	(* conversion string to value *)
		i:=1;
		(* read string line-->Group or NodeId *)
		sTmp:=T_Axis.T_FileObj.sData[i];
		iPosCarStart:=FIND(sTmp,':=')+2;
		iPosCarStop:=FIND(sTmp,';');
		IF ((iPosCarStart - 2) = 0) OR (iPosCarStop = 0) OR (iPosCarStart >= iPosCarStop) THEN xBusy:=FALSE;	xDone:=FALSE; xError:=TRUE; diErrorNr:=16#F100;	(* Wrong Syntax from Axis File *) RETURN; END_IF;
		T_Axis.T_Config_Gen.udiNC_TaskIdxGrp:=0;
		T_Axis.T_Config_Gen.udiNodeId:=STRING_TO_UDINT(MID(sTmp,iPosCarStop-iPosCarStart,iPosCarStart));
		i:=i+1;
		(* read string line-->ADS NetID *)
		sTmp:=T_Axis.T_FileObj.sData[i];
		iPosCarStart:=FIND(sTmp,':=')+2;
		iPosCarStop:=FIND(sTmp,';');
		IF ((iPosCarStart - 2) = 0) OR (iPosCarStop = 0) OR (iPosCarStart >= iPosCarStop) THEN xBusy:=FALSE;	xDone:=FALSE; xError:=TRUE; diErrorNr:=16#F100;	(* Wrong Syntax from Axis File *) RETURN; END_IF;
		T_Axis.T_Config_Gen.sServoNetId:='';
		T_Axis.T_Config_Gen.sAmsNetId:=MID(sTmp,iPosCarStop-iPosCarStart,iPosCarStart);
		i:=i+1;
		(* read string line-->DeviceName *)
		sTmp:=T_Axis.T_FileObj.sData[i];
		iPosCarStart:=FIND(sTmp,':=')+2;
   		iPosCarStop:=FIND(sTmp,';');
		IF ((iPosCarStart - 2) = 0) OR (iPosCarStop = 0) OR (iPosCarStart >= iPosCarStop) THEN xBusy:=FALSE;	xDone:=FALSE; xError:=TRUE; diErrorNr:=16#F100;	(* Wrong Syntax from Axis File *) RETURN; END_IF;
		T_Axis.T_Config_Gen.sFileNamePDOMapping:=MID(sTmp,iPosCarStop-iPosCarStart,iPosCarStart);
		i:=i+1;
		jj:=1;
		(* read string lines *)
		WHILE T_Axis.T_FileObj.sData[i] <> '' DO
			sTmp:=T_Axis.T_FileObj.sData[i];
			(* index group *)
			iPosCarStart:=FIND(sTmp,':=')+2;
			iPosCarStop:=FIND(sTmp,';');
			IF ((iPosCarStart - 2) = 0) OR (iPosCarStop = 0) OR (iPosCarStart >= iPosCarStop) THEN xBusy:=FALSE;	xDone:=FALSE; xError:=TRUE; diErrorNr:=16#F100;	(* Wrong Syntax from Axis File *) RETURN; END_IF;
			T_Axis.T_ParamFileObj[jj].udiIdxGroup:=	STRING_TO_UDINT(MID(sTmp,iPosCarStop-iPosCarStart,iPosCarStart))
											+ T_Axis.T_Config_Gen.udiNC_TaskIdxGrp;
			sTmp:=MID(sTmp,LEN(sTmp)-iPosCarStop, iPosCarStop+1);
			(* index offset *)
			iPosCarStart:=FIND(sTmp,':=')+2;
			iPosCarStop:=FIND(sTmp,';');
			IF ((iPosCarStart - 2) = 0) OR (iPosCarStop = 0) OR (iPosCarStart >= iPosCarStop) THEN xBusy:=FALSE;	xDone:=FALSE; xError:=TRUE; diErrorNr:=16#F100;	(* Wrong Syntax from Axis File *) RETURN; END_IF;
			T_Axis.T_ParamFileObj[jj].udiIndexOffset:=STRING_TO_UDINT(MID(sTmp,iPosCarStop-iPosCarStart,iPosCarStart));
			sTmp:=MID(sTmp,LEN(sTmp)-iPosCarStop, iPosCarStop+1);
			(* length value *)
			iPosCarStart:=FIND(sTmp,':=')+2;
			iPosCarStop:=FIND(sTmp,';');
			IF ((iPosCarStart - 2) = 0) OR (iPosCarStop = 0) OR (iPosCarStart >= iPosCarStop) THEN xBusy:=FALSE;	xDone:=FALSE; xError:=TRUE; diErrorNr:=16#F100;	(* Wrong Syntax from Axis File *) RETURN; END_IF;
			T_Axis.T_ParamFileObj[jj].udiLength:=STRING_TO_UDINT(MID(sTmp,iPosCarStop-iPosCarStart,iPosCarStart));
			sTmp:=MID(sTmp,LEN(sTmp)-iPosCarStop, iPosCarStop+1);
			(* value*)
			iPosCarStart:=FIND(sTmp,':=')+2;
			iPosCarStop:=FIND(sTmp,';');
			IF ((iPosCarStart - 2) = 0) OR (iPosCarStop = 0) OR (iPosCarStart >= iPosCarStop) THEN xBusy:=FALSE;	xDone:=FALSE; xError:=TRUE; diErrorNr:=16#F100;	(* Wrong Syntax from Axis File *) RETURN; END_IF;
			T_Axis.T_ParamFileObj[jj].lrReal:=UDINT_TO_REAL(STRING_TO_UDINT(MID(sTmp,iPosCarStop-iPosCarStart,iPosCarStart)));
			(* init existing line, erase text *)
			iPosCarStop:=FIND(T_Axis.T_FileObj.sData[i],'(');
			T_Axis.T_FileObj.sData[i]:=MID(T_Axis.T_FileObj.sData[i],iPosCarStop-1,1);
			(* next line *)
			i:=i+1;
			jj:=jj+1;
		END_WHILE
		(* init. next *)
		T_Axis.T_ParamFileObj[jj].udiIdxGroup:=0;
		T_Axis.T_ParamFileObj[jj].udiIndexOffset:=0;
		T_Axis.T_ParamFileObj[jj].udiLength:=0;
		T_Axis.T_ParamFileObj[jj].lrReal:=0;

		(* set flag done *)
		xBusy:=FALSE;
		xDone:=TRUE;
END_FUNCTION_BLOCK

(* POU FB_HARDWARE/FB_CONVERT_AXISPARAMETER, ST *)
FUNCTION_BLOCK FB_CONVERT_AXISPARAMETER
VAR_INPUT
	xStart:BOOL;
END_VAR
VAR_IN_OUT
	T_Axis:ST_AXIS;
END_VAR
VAR_OUTPUT
	xDone:BOOL;
	xBusy:BOOL;
	xError:BOOL;
	diErrorNr:DINT;
END_VAR
VAR
(* trigger *)
	RisingEdgeStart:R_TRIG;
(* variable *)
	i: INT;
	iPosCarStart,iPosCarStop:INT;
	iStepConvertValueString:INT;
(* tmp variable *)
	sTmp:STRING(255);
	jj: INT;
END_VAR
(****************************************************************************************************************************************************)
(***********                                    This Functionblock convert the axis parameter for the EcoStep drive                                       ************)
(****************************************************************************************************************************************************)
(* wait start *)
	RisingEdgeStart(CLK:=xStart);
	IF RisingEdgeStart.Q THEN
	(* init. varaible *)
		iStepConvertValueString:=1;
		xDone:=FALSE;
	(*activ busy flag*)
		xBusy:=TRUE;
		xError:=FALSE;
		diErrorNr:=0;
	END_IF

(* test if activ *)
	IF NOT(xBusy) THEN
	(* exit FB *)
		RETURN;
	END_IF

	(* conversion string to value *)
		i:=1;
		(* read string line-->Group or NodeId *)
		sTmp:=T_Axis.T_FileObj.sData[i];
		iPosCarStart:=FIND(sTmp,':=')+2;
		iPosCarStop:=FIND(sTmp,';');
		IF ((iPosCarStart - 2) = 0) OR (iPosCarStop = 0) OR (iPosCarStart >= iPosCarStop) THEN xBusy:=FALSE;	xDone:=FALSE; xError:=TRUE; diErrorNr:=16#F100;	(* Wrong Syntax from Axis File *) RETURN; END_IF;
		T_Axis.T_Config_Gen.udiNC_TaskIdxGrp:=0;
		T_Axis.T_Config_Gen.udiNodeId:=STRING_TO_UDINT(MID(sTmp,iPosCarStop-iPosCarStart,iPosCarStart));
		i:=i+1;
		(* read string line-->ADS NetID *)
		sTmp:=T_Axis.T_FileObj.sData[i];
		iPosCarStart:=FIND(sTmp,':=')+2;
		iPosCarStop:=FIND(sTmp,';');
		IF ((iPosCarStart - 2) = 0) OR (iPosCarStop = 0) OR (iPosCarStart >= iPosCarStop) THEN xBusy:=FALSE;	xDone:=FALSE; xError:=TRUE; diErrorNr:=16#F100;	(* Wrong Syntax from Axis File *) RETURN; END_IF;
		T_Axis.T_Config_Gen.sServoNetId:='';
		T_Axis.T_Config_Gen.sAmsNetId:=MID(sTmp,iPosCarStop-iPosCarStart,iPosCarStart);
		i:=i+1;
		(* read string line-->DeviceName *)
		sTmp:=T_Axis.T_FileObj.sData[i];
		iPosCarStart:=FIND(sTmp,':=')+2;
   		iPosCarStop:=FIND(sTmp,';');
		IF ((iPosCarStart - 2) = 0) OR (iPosCarStop = 0) OR (iPosCarStart >= iPosCarStop) THEN xBusy:=FALSE;	xDone:=FALSE; xError:=TRUE; diErrorNr:=16#F100;	(* Wrong Syntax from Axis File *) RETURN; END_IF;
		T_Axis.T_Config_Gen.sDeviceFileName:=MID(sTmp,iPosCarStop-iPosCarStart,iPosCarStart);
		i:=i+1;
		(* read string line-->Scalefactor *)
		sTmp:=T_Axis.T_FileObj.sData[i];
		iPosCarStart:=FIND(sTmp,':=')+2;
   		iPosCarStop:=FIND(sTmp,';');
		IF ((iPosCarStart - 2) = 0) OR (iPosCarStop = 0) OR (iPosCarStart >= iPosCarStop) THEN xBusy:=FALSE;	xDone:=FALSE; xError:=TRUE; diErrorNr:=16#F100;	(* Wrong Syntax from Axis File *) RETURN; END_IF;
		T_Axis.T_CtrleSingle.lrScaleFactor:=STRING_TO_LREAL(MID(sTmp,iPosCarStop-iPosCarStart,iPosCarStart));
		i:=i+1;
		(* read string line-->GearRatioFactor  *)
		sTmp:=T_Axis.T_FileObj.sData[i];
		iPosCarStart:=FIND(sTmp,':=')+2;
   		iPosCarStop:=FIND(sTmp,';');
		IF ((iPosCarStart - 2) = 0) OR (iPosCarStop = 0) OR (iPosCarStart >= iPosCarStop) THEN xBusy:=FALSE;	xDone:=FALSE; xError:=TRUE; diErrorNr:=16#F100;	(* Wrong Syntax from Axis File *) RETURN; END_IF;
		T_Axis.T_CtrleSingle.lrGearRatioFactor:=STRING_TO_LREAL(MID(sTmp,iPosCarStop-iPosCarStart,iPosCarStart));
		i:=i+1;
		(* read string line-->GearRatioDivider *)
		sTmp:=T_Axis.T_FileObj.sData[i];
		iPosCarStart:=FIND(sTmp,':=')+2;
   		iPosCarStop:=FIND(sTmp,';');
		IF ((iPosCarStart - 2) = 0) OR (iPosCarStop = 0) OR (iPosCarStart >= iPosCarStop) THEN xBusy:=FALSE;	xDone:=FALSE; xError:=TRUE; diErrorNr:=16#F100;	(* Wrong Syntax from Axis File *) RETURN; END_IF;
		T_Axis.T_CtrleSingle.lrGearRatioDivider:=STRING_TO_LREAL(MID(sTmp,iPosCarStop-iPosCarStart,iPosCarStart));
		IF (T_Axis.T_CtrleSingle.lrGearRatioFactor <> 0) AND (T_Axis.T_CtrleSingle.lrGearRatioDivider <> 0) THEN
			T_Axis.T_CtrleSingle.lrGearRatio:=T_Axis.T_CtrleSingle.lrGearRatioFactor/T_Axis.T_CtrleSingle.lrGearRatioDivider;
		ELSE
			T_Axis.T_CtrleSingle.lrGearRatio:=1;
		END_IF;
		i:=i+1;
		jj:=1;
		(* read string lines *)
		WHILE T_Axis.T_FileObj.sData[i] <> '' DO
			sTmp:=T_Axis.T_FileObj.sData[i];
			(* index group *)
			iPosCarStart:=FIND(sTmp,':=')+2;
			iPosCarStop:=FIND(sTmp,';');
			IF ((iPosCarStart - 2) = 0) OR (iPosCarStop = 0) OR (iPosCarStart >= iPosCarStop) THEN xBusy:=FALSE;	xDone:=FALSE; xError:=TRUE; diErrorNr:=16#F100;	(* Wrong Syntax from Axis File *) RETURN; END_IF;
			T_Axis.T_ParamFileObj[jj].udiIdxGroup:=	STRING_TO_UDINT(MID(sTmp,iPosCarStop-iPosCarStart,iPosCarStart))
											+ T_Axis.T_Config_Gen.udiNC_TaskIdxGrp;
			sTmp:=MID(sTmp,LEN(sTmp)-iPosCarStop, iPosCarStop+1);
			(* index offset *)
			iPosCarStart:=FIND(sTmp,':=')+2;
			iPosCarStop:=FIND(sTmp,';');
			IF ((iPosCarStart - 2) = 0) OR (iPosCarStop = 0) OR (iPosCarStart >= iPosCarStop) THEN xBusy:=FALSE;	xDone:=FALSE; xError:=TRUE; diErrorNr:=16#F100;	(* Wrong Syntax from Axis File *) RETURN; END_IF;
			T_Axis.T_ParamFileObj[jj].udiIndexOffset:=STRING_TO_UDINT(MID(sTmp,iPosCarStop-iPosCarStart,iPosCarStart));
			sTmp:=MID(sTmp,LEN(sTmp)-iPosCarStop, iPosCarStop+1);
			(* length value *)
			iPosCarStart:=FIND(sTmp,':=')+2;
			iPosCarStop:=FIND(sTmp,';');
			IF ((iPosCarStart - 2) = 0) OR (iPosCarStop = 0) OR (iPosCarStart >= iPosCarStop) THEN xBusy:=FALSE;	xDone:=FALSE; xError:=TRUE; diErrorNr:=16#F100;	(* Wrong Syntax from Axis File *) RETURN; END_IF;
			T_Axis.T_ParamFileObj[jj].udiLength:=STRING_TO_UDINT(MID(sTmp,iPosCarStop-iPosCarStart,iPosCarStart));
			sTmp:=MID(sTmp,LEN(sTmp)-iPosCarStop, iPosCarStop+1);
			(* value*)
			iPosCarStart:=FIND(sTmp,':=')+2;
			iPosCarStop:=FIND(sTmp,';');
			IF ((iPosCarStart - 2) = 0) OR (iPosCarStop = 0) OR (iPosCarStart >= iPosCarStop) THEN xBusy:=FALSE;	xDone:=FALSE; xError:=TRUE; diErrorNr:=16#F100;	(* Wrong Syntax from Axis File *) RETURN; END_IF;
			T_Axis.T_ParamFileObj[jj].lrReal:=UDINT_TO_REAL(STRING_TO_UDINT(MID(sTmp,iPosCarStop-iPosCarStart,iPosCarStart)));
			(* init existing line, erase text *)
			iPosCarStop:=FIND(T_Axis.T_FileObj.sData[i],'(');
			T_Axis.T_FileObj.sData[i]:=MID(T_Axis.T_FileObj.sData[i],iPosCarStop-1,1);
			(* next line *)
			i:=i+1;
			jj:=jj+1;
		END_WHILE
		(* init. next *)
		T_Axis.T_ParamFileObj[jj].udiIdxGroup:=0;
		T_Axis.T_ParamFileObj[jj].udiIndexOffset:=0;
		T_Axis.T_ParamFileObj[jj].udiLength:=0;
		T_Axis.T_ParamFileObj[jj].lrReal:=0;

		(* set flag done *)
		xBusy:=FALSE;
		xDone:=TRUE;
END_FUNCTION_BLOCK

(* POU FB_HARDWARE/FCT_GET_AXIS_ERROR, ST *)
FUNCTION FCT_GET_AXIS_ERROR : UDINT
VAR_INPUT
	dwInputBitStructError:DWORD;
END_VAR
VAR
	udiTmpErrorID:UDINT;
END_VAR
(****************************************************************************************************************************************************)
(***********                                             This Functionblock read the Axis error of the EcoStep drive                                                ************)
(****************************************************************************************************************************************************)
udiTmpErrorID:=0;
IF GETBIT32(dwInputBitStructError,0) THEN
	udiTmpErrorID:=16#F801;	(* Interne Ursache, darf niemals auftreten *)
END_IF;
IF GETBIT32(dwInputBitStructError,1) THEN
	udiTmpErrorID:=16#F802;	(* Interne Ursache, darf niemals auftreten *)
END_IF;
IF GETBIT32(dwInputBitStructError,2) THEN
	udiTmpErrorID:=16#F803;	(* Antivalenzfehler der Motorencodersignale (auf Drahtbruch beim Encoder an X8 prüfen) *)
END_IF;
IF GETBIT32(dwInputBitStructError,3) THEN
	udiTmpErrorID:=16#F804;	(* Encoder Zählfehler, >+/-4 inc, Encoderscheibe beschädigt oder verspannt *)
END_IF;
IF GETBIT32(dwInputBitStructError,4) THEN
	udiTmpErrorID:=16#F805;	(* Master Encoder X7 Zählfehler, >+/-4 inc, Encoderscheibe beschädigt oder verspannt *)
END_IF;
IF GETBIT32(dwInputBitStructError,5) THEN
	udiTmpErrorID:=16#F806;	(* Kühlkörpertemperatur zu hoch (> 80°) *)
END_IF;
IF GETBIT32(dwInputBitStructError,6) THEN
	udiTmpErrorID:=16#F807;	(* Unterspannung (<18V) der +24V Logikversorgung *)
END_IF;
IF GETBIT32(dwInputBitStructError,7) THEN
	udiTmpErrorID:=16#F808;	(* Überspannung X10 (>180V) der Leistungsversorgung DC_BUS (Netzteil prüfen;Rückspeisung beachten!) *)
END_IF;
IF GETBIT32(dwInputBitStructError,8) THEN
	udiTmpErrorID:=16#F809;	(* Unterspannung X10 (<24V) der Leistungsversorgung DC_BUS (Netzteil prüfen!) *)
END_IF;
IF GETBIT32(dwInputBitStructError,9) THEN
	udiTmpErrorID:=16#F80A;	(* Kurzschluss in Motorphase A *)
END_IF;
IF GETBIT32(dwInputBitStructError,10) THEN
	udiTmpErrorID:=16#F80B;	(* Kurzschluss in Motorphase B *)
END_IF;
IF GETBIT32(dwInputBitStructError,11) THEN
	udiTmpErrorID:=16#F80C;	(* Kurzschluss eines digitalen Ausgangs während Antrieb eingeschaltet war *)
END_IF;
IF GETBIT32(dwInputBitStructError,12) THEN
	udiTmpErrorID:=16#F80D;	(* Digital-Eingang "ENABLE" wurde auf Low-Pegel gesetzt während der Antrieb eingeschaltet war *)
END_IF;
IF GETBIT32(dwInputBitStructError,13) THEN
	udiTmpErrorID:=16#F80E;	(* Max. Schleppfehler überschritten (im Positioniermodus) *)
END_IF;
IF GETBIT32(dwInputBitStructError,14) THEN
	udiTmpErrorID:=16#F80F;	(* Drehzahl zu hoch, Regler kann Encoder nicht mehr auslesen (>4MHz) *)
END_IF;
IF GETBIT32(dwInputBitStructError,15) THEN
	udiTmpErrorID:=16#F810;	(* Kommutierung nicht gefunden *)
END_IF;
IF GETBIT32(dwInputBitStructError,16) THEN
	udiTmpErrorID:=16#F811;	(* CAN-Kommunikation unterbrochen bei Node Guarding *)
END_IF;
IF GETBIT32(dwInputBitStructError,17) THEN
	udiTmpErrorID:=16#F812;	(* I^2t- Überwachung ausgelöst (Stromgrenze) *)
END_IF;
FCT_GET_AXIS_ERROR:=udiTmpErrorID;
END_FUNCTION

(* POU FB_HARDWARE/FBHW_AXIS_LIVEVALUES_ECOSTEP, ST *)
FUNCTION_BLOCK FBHW_AXIS_LIVEVALUES_ECOSTEP
VAR_INPUT
	iTypAxis:INT;	(* 1:ToolRotation, 2:ToolFeed, 3:GrindFeed *)
	rPrismaFactor:REAL;
	xMicroRodActive: BOOL;		(* choice of the machine MicroWire or MicroRod *)
END_VAR
VAR_IN_OUT
	T_Axis:ST_AXIS;
END_VAR
VAR_OUTPUT
END_VAR
VAR
	rActualCurrent: REAL;
	rMultiplier: REAL;
	TONCheckTime: TON;
END_VAR
(****************************************************************************************************************************************************)
(***********                                    This Functionblock read the actual value from the EcoStep drive                                               ************)
(****************************************************************************************************************************************************)
(* Monitoring of the Internal Limit is Active *)
(* IF ((iTypAxis = 4) OR (iTypAxis = 5)) AND (T_Axis.T_Config_ObjFileValue.xSWLimitPos OR T_Axis.T_Config_ObjFileValue.xSWLimitNeg) THEN*)
IF (	T_Axis.T_Config_ObjFileValue.xSWLimitPos OR T_Axis.T_Config_ObjFileValue.xSWLimitNeg OR T_Axis.T_Config_ObjFileValue.xSWLimitPos OR	T_Axis.T_Config_ObjFileValue.xHWLimitNeg ) THEN	(* Only for ToolFeeder and GrindFeeder *)
	TONCheckTime(IN:=GETBIT32(T_Axis.T_TxPdoParameter.uiStatusWord,11),PT:=T#1000ms);
	IF TONCheckTime.Q  THEN			(* check if the internal limit bit for the statusword is set *)
		IF GETBIT32(T_Axis.T_TxPdoParameter.udiDigitalInput,21) THEN	(* DIN 6 form Ecostep Drive *)
			T_Axis.T_CtrleSingle.xHWLimitPos:=TRUE;
			T_Axis.T_CtrleSingle.xSWLimitPos:=FALSE;
		ELSE
			T_Axis.T_CtrleSingle.xHWLimitPos:=FALSE;
			T_Axis.T_CtrleSingle.xSWLimitPos:=TRUE;
		END_IF;
		IF GETBIT32(T_Axis.T_TxPdoParameter.udiDigitalInput,22) THEN	(* DIN 7 from Ecostep Drive *)
			T_Axis.T_CtrleSingle.xHWLimitNeg:=TRUE;
			T_Axis.T_CtrleSingle.xSWLimitNeg:=FALSE;
		ELSE
			T_Axis.T_CtrleSingle.xHWLimitNeg:=FALSE;
			T_Axis.T_CtrleSingle.xSWLimitNeg:=TRUE;
		END_IF;
	ELSE
		IF GETBIT32(T_Axis.T_TxPdoParameter.udiDigitalInput,21) THEN	(* DIN 6 form Ecostep Drive *)
			T_Axis.T_CtrleSingle.xHWLimitPos:=TRUE;
		ELSE
			T_Axis.T_CtrleSingle.xHWLimitPos:=FALSE;
		END_IF;
		IF GETBIT32(T_Axis.T_TxPdoParameter.udiDigitalInput,22) THEN	(* DIN 7 from Ecostep Drive *)
			T_Axis.T_CtrleSingle.xHWLimitNeg:=TRUE;
		ELSE
			T_Axis.T_CtrleSingle.xHWLimitNeg:=FALSE;
		END_IF;
		T_Axis.T_CtrleSingle.xSWLimitPos:=FALSE;
		T_Axis.T_CtrleSingle.xSWLimitNeg:=FALSE;
	END_IF;
ELSE
	T_Axis.T_CtrleSingle.xHWLimitPos:=FALSE;
	T_Axis.T_CtrleSingle.xSWLimitPos:=FALSE;
	T_Axis.T_CtrleSingle.xHWLimitNeg:=FALSE;
	T_Axis.T_CtrleSingle.xSWLimitNeg:=FALSE;
	TONCheckTime(IN:=FALSE);
END_IF;

(* Monitoring of the actual position of the Ecostep Drive in technical unit *)
IF xMicroRodActive THEN
	IF (T_Axis.T_CtrleSingle.lrScaleFactor <> 0.0) THEN
		IF (iTypAxis <> 5) THEN	(* No GrindFeed Axis *)
			T_Axis.T_LiveValue.lrActualPosition:=DINT_TO_LREAL(T_Axis.T_TxPdoParameter.diActualPosition) / T_Axis.T_CtrleSingle.lrScaleFactor;
			T_Axis.T_LiveValue.lrActualPositionRelativ:=LMOD ( DINT_TO_LREAL(T_Axis.T_TxPdoParameter.diActualPosition) / T_Axis.T_CtrleSingle.lrScaleFactor, 360.0);
		ELSE
			IF (rPrismaFactor <> 0.0) THEN
				T_Axis.T_LiveValue.lrActualPosition:=DINT_TO_LREAL(T_Axis.T_TxPdoParameter.diActualPosition) / T_Axis.T_CtrleSingle.lrScaleFactor / rPrismaFactor;
			END_IF;
		END_IF;
	END_IF;
ELSE
	IF (T_Axis.T_CtrleSingle.lrScaleFactor <> 0.0) THEN
		IF (iTypAxis <> 5) THEN	(* No GrindFeed Axis *)
			T_Axis.T_LiveValue.lrActualPosition:=DINT_TO_LREAL(T_Axis.T_TxPdoParameter.diActualPosition) / T_Axis.T_CtrleSingle.lrScaleFactor;
		ELSE
			IF (rPrismaFactor <> 0.0) THEN
				T_Axis.T_LiveValue.lrActualPosition:=DINT_TO_LREAL(T_Axis.T_TxPdoParameter.diActualPosition) / T_Axis.T_CtrleSingle.lrScaleFactor / rPrismaFactor;
			END_IF;
		END_IF;
	END_IF;
END_IF
(* Monitoring of the actual position of the Ecostep Drive in increments *)
T_Axis.T_LiveValue.lrActualPositionNotModulo:=DINT_TO_LREAL(T_Axis.T_TxPdoParameter.diActualPosition);

(* Monitoring of the actual speed of the Ecostep Drive *)
IF (iTypAxis = 1) OR (iTypAxis = 2) OR (iTypAxis = 3) THEN	(* rotative motion *)
	IF (T_Axis.T_CtrleSingle.lrScaleFactor <> 0.0) THEN
		T_Axis.T_LiveValue.lrActualVelocity:=((DINT_TO_LREAL(T_Axis.T_TxPdoParameter.diActualVelocity) * 60.0)/(T_Axis.T_CtrleSingle.lrScaleFactor*64.0))/360.0;
	END_IF;
END_IF;
IF (iTypAxis = 4) OR (iTypAxis = 5) THEN	(* linear motion *)
	IF (T_Axis.T_CtrleSingle.lrScaleFactor <> 0.0) THEN
		T_Axis.T_LiveValue.lrActualVelocity:=ABS(DINT_TO_LREAL(T_Axis.T_TxPdoParameter.diActualVelocity)/(T_Axis.T_CtrleSingle.lrScaleFactor*64.0));
	END_IF;
END_IF;

(* Monitoring of the actual torque, 23S21 Motor constant of the Motortorque: 0.16Nm/A, max servodrive current 12A *)
IF (T_Axis.T_TxPdoParameter.iActualCurrent < 0) THEN
	rActualCurrent:=ABS(T_Axis.T_TxPdoParameter.iActualCurrent);
	rMultiplier:=-1.0;
ELSE
	rActualCurrent:=T_Axis.T_TxPdoParameter.iActualCurrent;
	rMultiplier:=1.0;
END_IF;
T_Axis.T_LiveValue.uiActualTorque:=REAL_TO_UINT(((12.0/2047.0) * rActualCurrent * 0.16) * 1000.0);	(* convert from Nm in mNm-->Absolut value *)
T_Axis.T_LiveValue.diActualTorqueCalc:=REAL_TO_DINT(((12.0/2047.0) * rActualCurrent * rMultiplier * 0.16) * 1000.0);	(* convert from Nm in mNm, positive and negative value *)

(* Monitoring of the statusword *)
T_Axis.T_LiveValue.dwState:=UINT_TO_DWORD(T_Axis.T_TxPdoParameter.uiStatusWord);
END_FUNCTION_BLOCK

(* POU FB_HARDWARE/FBHW_AXIS_SINGLE_BECKHOFF, ST *)
FUNCTION_BLOCK FBHW_AXIS_SINGLE_BECKHOFF
VAR_INPUT
	xHWLimitPos:BOOL:=FALSE;
	xHWLimitNeg:BOOL:=FALSE;
	xRefHoming:BOOL:=FALSE;
END_VAR
VAR_OUTPUT
END_VAR
VAR_IN_OUT
	T_Axis:ST_AXIS;
	T_AxisRefIn:NCTOPLC_AXLESTRUCT;
	T_AxisRefOut:PLCTONC_AXLESTRUCT;
	T_HDD:ST_HDD;
END_VAR
VAR
(* Axis function block *)
	fbAxisReset:MC_Reset;
	fbAxisPower:MC_Power;
	fbAxisStop:MC_Stop;
	fbAxisMoveVelocity:MC_MoveVelocity;
	fbAxisMoveAbsolute:MC_MoveAbsolute;
	fbAxisMoveRelative:MC_MoveRelative;
	fbAxisMoveModulo:MC_MoveModulo;
	fbAxisHoming:MC_Home;
	fbAxisSetOverride:MC_SetOverride;
	fbAxisSetPosition:MC_SetActualPosition;
	fbAxisNewPosAndVel:MC_NewPosAndVelo;
	fbAxisSetReferenceFlag:MC_SetReferenceFlag;
	fbDefaultAxisPara:FB_DEFAULT_AXISVALUE;
	fbAdsWrite:ADSWRITE;
	fbADS_ReadWriteString:ADSRDWRTEX;
	fb_ConvertParaAxis:FB_CONVERT_PARA_AXIS;
	fbExtSetPointGenDisable:MC_ExtSetPointGenDisable;
	fbExtSetPointGenEnable:MC_ExtSetPointGenEnable;

(* variable *)
	xConfirmResetFB:BOOL:=FALSE;
	xResetAxis:BOOL:=FALSE;
	xReadFile:BOOL:=FALSE;
	xPowerOn:BOOL:=FALSE;
	xPowerOff:BOOL:=FALSE;
	xStop:BOOL:=FALSE;
	xMoveVel:BOOL:=FALSE;
	iDirectionVel:INT:=1;
	rVelocity:REAL:=0;
	xMoveAbs:BOOL:=FALSE;
	xMoveRel:BOOL:=FALSE;
	xMoveModulo:BOOL:=FALSE;
	xHoming:BOOL:=FALSE;
	xOverride:BOOL:=FALSE;
	xSetPosition:BOOL:=FALSE;
	xNewVelocity:BOOL:=FALSE;
	xNewPosition:BOOL:=FALSE;
	xCalcAngleRefIndex: BOOL:=FALSE;
	xSetReferenceFlag:BOOL:=FALSE;
	xResetReferenceFlag:BOOL:=FALSE;
	xDefaultAxisParameter:BOOL:=FALSE;
	xSendAxisParameter:BOOL:=FALSE;
	iPtrAxisParameter:INT:=0;
	xSendAxisString:BOOL:=FALSE;
	sSendAxis:STRING:='';
	sReturnAxis:STRING:='';
	iStepSendPara:INT:=0;
	xRestoreAxisPower:BOOL:=FALSE;
	iStepFile:INT:=0;
	xWriteFile: BOOL:=FALSE;
	xCtrlePositionOn:BOOL:=FALSE;
	xCtrlePositionOff:BOOL:=FALSE;
	xOscillation:BOOL:=FALSE;
	iStepOsc:INT:=0;
	iOscCounter:INT:=0;
	iStepResetFB:INT:=0;
	dwOldOverride:DWORD:=100;
	lrOverrideVel:LREAL;
(* timer *)
	TimerOutSendPara:TON;
	TimerFileLocked:TON;

(* trigger *)
	RisingEdgeStop:R_TRIG;
	RisingEdgeResetFB:R_TRIG;
	RisingEdgeExecute:R_TRIG;
	RisingEdgePowerOn:R_TRIG;
	RisingEdgePowerOff:R_TRIG;

(* Temp variable *)
	xTmp:BOOL:=FALSE;
	i:INT;
	wTmp:WORD:=0;
	dwTmp:DWORD:=0;
	dwAdrVar:DWORD:=0;
	sTmp:STRING(255);
	rTmpFrequence:REAL;
	lrTmpVelocity:LREAL;
	TimerCommTimeLeft:TON;
	xStartTimerComm:BOOL:=FALSE;
	tTimeCommLeft:TIME;
	TimerCommTimeLeft1:TON;
	xStartTimerComm1:BOOL:=FALSE;
	tTimeCommLeft1:TIME;
	sDeleteData: ARRAY[1..csiMaxAxisFileObj] OF STRING(120);
	xMovement: BOOL;
	xNoHWError: BOOL;
	iStepCalcRefIndex: INT;
	xCheckRefState: BOOL;
	iTmpFctNr: INT;
	lrTechUnitPerMotorTurn: LREAL;	(* Gilt nur für das Aufsuchen des Reference Index-->Die Technische Einheit muss angegeben werden, damit eine Motorrotation durchgeführt werden kann z.B. 2.5mm/U_Motor  oder 30Grad/U_Motor*)
	xSendBlock: BOOL;
	lrCapturePosition: LREAL;
END_VAR
(****************************************************************************************************************************************************)
(***********                                               This Functionblock is the driver for the Beckhoff Axis                                                           ************)
(****************************************************************************************************************************************************)
(* Test Timer PUM *)
TimerCommTimeLeft(IN:=xStartTimerComm,PT:=T#99999s);
TimerCommTimeLeft1(IN:=xStartTimerComm1,PT:=T#99999s);
(* reset block function *)
	RisingEdgeResetFB(CLK:=T_Axis.T_CtrleSingle.xReset);
	IF RisingEdgeResetFB.Q THEN
	(* Init. block function *)
		fbAxisReset(Execute:=FALSE, Axis:=T_AxisRefIn);
		fbAxisPower(	Enable:=FALSE,
					AxisRefIn:=T_AxisRefIn,
					AxisRefOut:=T_AxisRefOut);
		fbAxisStop(Execute:=FALSE, Axis:=T_AxisRefIn);
		fbAxisMoveVelocity(Execute:=FALSE, Axis:=T_AxisRefIn);
		fbAxisMoveAbsolute(Execute:=FALSE, Axis:=T_AxisRefIn);
		fbAxisMoveModulo(Execute:=FALSE, Axis:=T_AxisRefIn);
		fbAxisMoveRelative(Execute:=FALSE, Axis:=T_AxisRefIn);
		fbAxisHoming(	Execute:=FALSE,
						Axis:=T_AxisRefIn,
						AxisOut:=T_AxisRefOut);
		fbAxisSetOverride(Execute:=FALSE,
						AxisRefIn:=T_AxisRefIn,
						AxisRefOut:=T_AxisRefOut);
		fbAxisSetPosition(	Execute:=FALSE, Axis:=T_AxisRefIn);
		fbAxisNewPosAndVel(	Execute:=FALSE,
							Axis:=T_AxisRefIn);
		fbAdsWrite(WRITE:=FALSE);
		fbADS_ReadWriteString(WRTRD:=FALSE);
	(* timer *)
		TimerOutSendPara(IN:=TRUE,PT:=T#1ms);
	(* Init. variable *)
		xResetAxis:=FALSE;
		xReadFile:=FALSE;
		xPowerOn:=FALSE;
		xPowerOff:=FALSE;
		xStop:=FALSE;
		xMoveVel:=FALSE;
		iDirectionVel:=1;
		rVelocity:=0;
		xMoveAbs:=FALSE;
		xMoveRel:=FALSE;
		xMoveModulo:=FALSE;
		xHoming:=FALSE;
		xOverride:=FALSE;
		xSetPosition:=FALSE;
		xNewVelocity:=FALSE;
		xNewPosition:=FALSE;
		xCalcAngleRefIndex:=FALSE;
		xSetReferenceFlag:=FALSE;
		xResetReferenceFlag:=FALSE;
		xDefaultAxisParameter:=FALSE;
		xSendAxisParameter:=FALSE;
		iPtrAxisParameter:=1;
		xSendAxisString:=FALSE;
		iStepSendPara:=0;
		xRestoreAxisPower:=FALSE;
		xWriteFile:=FALSE;
		iStepFile:=0;
		xCtrlePositionOn:=FALSE;
		xCtrlePositionOff:=FALSE;
		xOscillation:=FALSE;
		iStepOsc:=0;
		iOscCounter:=0;
		iStepCalcRefIndex:=0;
	(* int. structure *)
		T_Axis.T_CtrleSingle.dwOverride:=100;
		T_Axis.T_CtrleSingle.iFunction:=0;
		T_Axis.T_CtrleSingle.xDone:=FALSE;
		T_Axis.T_CtrleSingle.xErr:=FALSE;
		T_Axis.T_CtrleSingle.udiErrorID:=0;
		T_Axis.T_CtrleSingle.xPower:=FALSE;
		T_Axis.T_CtrleSingle.xReady:=FALSE;
		T_Axis.T_CtrleSingle.xNotMoving:=FALSE;
		T_Axis.T_CtrleSingle.xRef:=FALSE;
		T_Axis.T_CtrleSingle.xSlave:=FALSE;
		T_Axis.T_CtrleSingle.xConstantVel:=FALSE;
		T_Axis.T_CtrleSingle.xBusyNewPosAndVel:=FALSE;
		T_Axis.T_CtrleSingle.xDriveTorque:=FALSE;
		(* set flag done *)
		xConfirmResetFB:=TRUE;
		(* disable status flag *)
		T_Axis.T_CtrleSingle.xDone:=FALSE;
		T_Axis.T_CtrleSingle.xErr:=FALSE;
		T_Axis.T_CtrleSingle.udiErrorID:=0;
		(* exit function bloc *)
		(* Test Timer PUM *)
		xStartTimerComm:=FALSE;
		xStartTimerComm1:=FALSE;
		RETURN;
	ELSE
		IF xConfirmResetFB THEN
		(* confirm reset FB *)
			T_Axis.T_CtrleSingle.xDone:=TRUE;
			T_Axis.T_CtrleSingle.xErr:=FALSE;
			T_Axis.T_CtrleSingle.udiErrorID:=0;
			(* reset variable *)
			xConfirmResetFB:=FALSE;
		END_IF
	END_IF

(* return axis state *)
	T_Axis.T_CtrleSingle.xReady:=GETBIT32(T_AxisRefIn.nStateDWord,0);
	T_Axis.T_CtrleSingle.xRef:=GETBIT32(T_AxisRefIn.nStateDWord,1);
	T_Axis.T_CtrleSingle.xNotMoving:=GETBIT32(T_AxisRefIn.nStateDWord,2);
	T_Axis.T_CtrleSingle.xSlave:=GETBIT32(T_AxisRefIn.nStateDWord,5);
	T_Axis.T_CtrleSingle.xConstantVel:=GETBIT32(T_AxisRefIn.nStateDWord,12);
	T_Axis.T_CtrleSingle.xSpindleBlocked:=NOT(T_Axis.T_CtrleSingle.xNotMoving) AND (ABS(T_Axis.T_LiveValue.lrActualVelocity) = 0);
	IF GETBIT32(T_AxisRefIn.nStateDWord,31) THEN
	(* error servo *)
		T_Axis.T_CtrleSingle.xDone:=FALSE;
		T_Axis.T_CtrleSingle.xErr:=TRUE;
		T_Axis.T_CtrleSingle.udiErrorID:=T_AxisRefIn.nErrorCode;
	END_IF

(* Timer *)
	TimerOutSendPara(IN:=TRUE, PT:=T#10S);
	TimerFileLocked(IN:=TRUE, PT:=T#10S);

(* determin if SW limit detection is activ *)
	(* positiv limit *)
	T_Axis.T_CtrleSingle.xSWLimitPos:=FALSE;
	IF (T_AxisRefIn.nOpModeDWord AND 16#80000) = 16#80000 THEN
		IF T_Axis.T_LiveValue.lrActualPosition >= T_Axis.T_Config_ObjFileValue.lrSWLimitPos THEN
			T_Axis.T_CtrleSingle.xSWLimitPos:=TRUE;
		END_IF
	END_IF
	(* negativ limit *)
	T_Axis.T_CtrleSingle.xSWLimitNeg:=FALSE;
	IF (T_AxisRefIn.nOpModeDWord AND 16#40000) = 16#40000 THEN
		IF T_Axis.T_LiveValue.lrActualPosition <= T_Axis.T_Config_ObjFileValue.lrSWLimitNeg THEN
			T_Axis.T_CtrleSingle.xSWLimitNeg:=TRUE;
		END_IF
	END_IF

(* detection hardware limit *)
	(* positiv limit *)
	IF T_Axis.T_Config_Setting.xHardwareLimitPos THEN T_Axis.T_CtrleSingle.xHWLimitPos:=NOT(xHWLimitPos);
	ELSE T_Axis.T_CtrleSingle.xHWLimitPos:=FALSE; END_IF
	(* negativ limit *)
	IF T_Axis.T_Config_Setting.xHardwareLimitNeg THEN T_Axis.T_CtrleSingle.xHWLimitNeg:=NOT(xHWLimitNeg);
	ELSE T_Axis.T_CtrleSingle.xHWLimitNeg:=FALSE; END_IF

	(* monitor hardware limit *)
	RisingEdgeStop(CLK:=T_Axis.T_CtrleSingle.xHWLimitPos OR T_Axis.T_CtrleSingle.xHWLimitNeg);
	IF NOT(T_Axis.T_CtrleSingle.xNotMoving) THEN
		IF RisingEdgeStop.Q THEN
		(* set decceleration ramp and make a stop *)
			xStop:=TRUE;
			IF T_Axis.T_Config_Setting.lrHWLimitDecceleration <> 0 THEN
				T_Axis.T_CtrleSingle.lrDecceleration:=T_Axis.T_Config_Setting.lrHWLimitDecceleration;
			END_IF
		END_IF
	END_IF

(* detection start *)
	RisingEdgeExecute(CLK:=T_Axis.T_CtrleSingle.xExecute);
	IF RisingEdgeExecute.Q THEN
		RisingEdgeExecute(CLK:=FALSE);
		IF xStop AND (T_Axis.T_CtrleSingle.iFunction <> 1) THEN
		(* can not execute a function when 'Stop' activ, except 'Reset' *)
			T_Axis.T_CtrleSingle.xDone:=FALSE;
			T_Axis.T_CtrleSingle.xErr:=TRUE;
			T_Axis.T_CtrleSingle.udiErrorID:=16#F100;
			RETURN;
		END_IF
		CASE T_Axis.T_CtrleSingle.iFunction OF
		(* Reset *)
		1:	xResetAxis:=TRUE;
			iStepResetFB:=1;
			iTmpFctNr:=1;
		(* Init *)
		2:	xReadFile:=TRUE;
			iStepFile:=1;
			iTmpFctNr:=2;
		(* Power ON *)
		3:	IF NOT(xPowerOn) THEN
				xPowerOn:=TRUE;
				xPowerOff:=NOT(xPowerOn);
				iTmpFctNr:=3;
			ELSE
				T_Axis.T_CtrleSingle.xDone:=TRUE;
				T_Axis.T_CtrleSingle.xErr:= FALSE;
				T_Axis.T_CtrleSingle.udiErrorID:=16#0;
				iTmpFctNr:=3;
				RETURN;
			END_IF;
		(* Power Off *)
		4:	IF xPowerOn THEN
				xPowerOff:=TRUE;
				xPowerOn:=NOT(xPowerOff);
				iTmpFctNr:=4;
			ELSE
				T_Axis.T_CtrleSingle.xDone:=TRUE;
				T_Axis.T_CtrleSingle.xErr:= FALSE;
				T_Axis.T_CtrleSingle.udiErrorID:=16#0;
				iTmpFctNr:=4;
				RETURN;
			END_IF;
		(* Stop *)
		5: 	xStop:=TRUE;
			fbAxisStop(Execute:=FALSE, Axis:=T_AxisRefIn);
			xStartTimerComm1:=TRUE;
			iTmpFctNr:=5;
		(* Velocity *)
		6:	xMoveVel:=TRUE;
			iTmpFctNr:=6;
		(* Absolute *)
		7:	xMoveAbs:=TRUE;
			iTmpFctNr:=7;
		(* Relative *)
		8:	xMoveRel:=TRUE;
			iTmpFctNr:=8;
		(* homing *)
		9:	xHoming:=TRUE;
			iTmpFctNr:=9;
		(* override *)
		10:	xOverride:=TRUE;
			iTmpFctNr:=10;
		(* set position *)
		11:	xSetPosition:=TRUE;
			iTmpFctNr:=11;
		(* change current speed *)
		12:	xNewVelocity:=TRUE;
			T_Axis.T_CtrleSingle.xBusyNewPosAndVel:=TRUE;
			IF xMoveAbs OR xMoveRel OR xMoveModulo OR xOscillation THEN	(* Muss unterschieden werden können, ob Positionsfahrt oder Velocitymode ausgeführt wird *)
				xMovement:=TRUE;
			ELSE
				xMovement:=FALSE;
			END_IF;
			xStartTimerComm:=TRUE;
		(* Set reference flag *)
		13:	xSetReferenceFlag:=TRUE;
			iTmpFctNr:=13;
		(* reset reference flag *)
		14:	xResetReferenceFlag:=TRUE;
			iTmpFctNr:=14;
		(* control position On *)
		15:	xCtrlePositionOn:=TRUE;
			iTmpFctNr:=15;
		(* control position off *)
		16:	xCtrlePositionOff:=TRUE;
			iTmpFctNr:=16;
		(* oscillation *)
		17:	xOscillation:=TRUE;
			iTmpFctNr:=17;
		(* change position *)
		18:	xNewPosition:=TRUE;
			T_Axis.T_CtrleSingle.xBusyNewPosAndVel:=TRUE;
		(* calcultate angle between Reference Index and Reference Sensor *)
		19:	xCalcAngleRefIndex:=TRUE;
			iTmpFctNr:=19;
		(* Default parameter value *)
		20:	xDefaultAxisParameter:=TRUE;
			iTmpFctNr:=20;
		(* Send Parameter *)
		21: 	xSendAxisParameter:=TRUE;
			iPtrAxisParameter:=1;
			iStepSendPara:=1;
			(* copy parameter value *)
			fbDefaultAxisPara(xDefaultValue:=FALSE,T_Axis:=T_Axis);
			iTmpFctNr:=21;
		(* send string *)
		22: 	xSendAxisString:=TRUE;
			sSendAxis:='';
			sReturnAxis:='';
			iTmpFctNr:=22;
		(* save parameter to file *)
		23:	xWriteFile:=TRUE;
			iStepFile:=11;
			iTmpFctNr:=23;
		(* Move Modulo *)
		24:	xMoveModulo:=TRUE;
			iTmpFctNr:=24;
		ELSE
		(* function not implemented *)
			T_Axis.T_CtrleSingle.xDone:=FALSE;
			T_Axis.T_CtrleSingle.xErr:=TRUE;
			T_Axis.T_CtrleSingle.udiErrorID:=16#F000;
			(* Exit FB *)
			RETURN;
		END_CASE
		(* Init. variable *)
		T_Axis.T_CtrleSingle.xDone:=FALSE;
		T_Axis.T_CtrleSingle.xErr:=FALSE;
		T_Axis.T_CtrleSingle.udiErrorID:=0;
		(* init variable *)
		dwOldOverride:=16#FFFF;
		(* Exit FB *)
		RETURN;
	END_IF

(* Override *)
	IF dwOldOverride <>T_Axis.T_CtrleSingle.dwOverride THEN
		lrOverrideVel:=T_Axis.T_CtrleSingle.lrVelocity * T_Axis.T_CtrleSingle.dwOverride / 100;
		(* confirm velocity setting *)
		dwOldOverride:=T_Axis.T_CtrleSingle.dwOverride;
	END_IF

(* Reset function *)
	IF xResetAxis THEN
		CASE iStepResetFB OF
		(* check state *)
		1:	xRestoreAxisPower:=FALSE;
			IF xPowerOn THEN iStepResetFB:=10; ELSE iStepResetFB:=20; END_IF
		(* power off *)
		10:	xPowerOff:=TRUE;
			xPowerOn:=NOT(xPowerOff);
			xRestoreAxisPower:=TRUE;
			(* next step *)
			iStepResetFB:=20;
		(* wait power off flag *)
		20:	IF NOT(T_Axis.T_CtrleSingle.xPower) THEN
				fbAxisReset(Execute:=TRUE, Axis:=T_AxisRefIn);
				IF fbAxisReset.Done OR fbAxisReset.Error THEN
					 IF fbAxisReset.Error THEN
						T_Axis.T_CtrleSingle.xDone:=fbAxisReset.Done;
						T_Axis.T_CtrleSingle.xErr:= fbAxisReset.Error;
						T_Axis.T_CtrleSingle.udiErrorID:=fbAxisReset.ErrorID;
					ELSE
					(* activ stop *)
						xStop:=TRUE;
						(* flag reset off only if the power has not to be recovered *)
						IF NOT(xRestoreAxisPower) THEN xResetAxis:=FALSE; END_IF
					END_IF
					(* reset flag busy *)
					T_Axis.T_CtrleSingle.xBusyNewPosAndVel:=FALSE;
					(* init. FB reset *)
					fbAxisReset(Execute:=FALSE, Axis:=T_AxisRefIn);
					(* next step *)
					iStepResetFB:=30;
				END_IF
			END_IF
		(* wait stop done *)
		30:	IF NOT(xStop) THEN iStepResetFB:=40; END_IF
		(* set power on *)
		40:	xPowerOff:=FALSE;
			xPowerOn:=NOT(xPowerOff);
			(* next step *)
			iStepResetFB:=50;
		(* wait power on flag *)
		50:	IF T_Axis.T_CtrleSingle.xPower THEN
			(* confirm reset *)
				T_Axis.T_CtrleSingle.xDone:=TRUE;
				T_Axis.T_CtrleSingle.xErr:= FALSE;
				T_Axis.T_CtrleSingle.udiErrorID:=16#0;
				(* init. variable *)
				xResetAxis:=FALSE;
			END_IF
		END_CASE
	ELSE fbAxisReset(Execute:=FALSE, Axis:=T_AxisRefIn); END_IF

(* Initialisation function *)
	IF xReadFile OR xWriteFile THEN
		CASE iStepFile OF
		(* start timeout *)
		1:	TimerFileLocked(IN:=FALSE);
			T_Axis.T_FileObj.sData:=sDeleteData;
			(* next step *)
			iStepFile:=iStepFile+1;
		(* start read *)
		2:	IF T_HDD.T_Ctrle.xDone AND NOT(T_HDD.T_Ctrle.xLocked) THEN
			(* activ read axis nc parameter *)
				T_HDD.T_Ctrle.xExecute:=TRUE;
				T_HDD.T_Ctrle.xLocked :=TRUE;
				T_HDD.T_Ctrle.iFunction:=1;
				sTmp:=CONCAT(cssRootPLC,'\Hard Disk\Bore800\Axis\File\');
				sTmp:=CONCAT(sTmp, T_Axis.T_Config_Gen.sDeviceFileName);
				T_HDD.T_File.sPathAndFileName:=CONCAT(sTmp,'.txt');
				(* next step *)
				iStepFile:=iStepFile+1;
			ELSE
			(* activ error if time out done, HDD not ready *)
				IF TimerFileLocked.Q THEN
					 iStepFile:=91;
				END_IF
			END_IF
		(* wait done or error *)
		3:	IF T_HDD.T_Ctrle.xDone OR T_HDD.T_Ctrle.xErr THEN
				IF T_HDD.T_Ctrle.xErr  THEN
				(* active step error *)
					iStepFile:=93;
				ELSE
				(* next step, init convert value *)
					iStepFile:=iStepFile+1;
					(* copy data from file *)
					i:=1;
					WHILE T_HDD.T_Data.sData[i] <> '' AND i <=csiMaxAxisFileObj AND i <= csiMaxFileLine DO
						T_Axis.T_FileObj.sData[i]:=T_HDD.T_Data.sData[i];
						i:=i+1;
					END_WHILE
					(* erase last line +1 *)
					IF i < csiMaxAxisFileObj THEN T_Axis.T_FileObj.sData[i+1]:=''; END_IF
				END_IF
			END_IF
		(* init. convert *)
		4:	fb_ConvertParaAxis(	xStart:=FALSE,
								T_Axis:=T_Axis);
			(* next step, convert value *)
			iStepFile:=iStepFile+1;
		(* convert value *)
		5:	fb_ConvertParaAxis(	xStart:=TRUE,
								iConversion:=0,
									sDeviceName:='Beckhoff',
									T_Axis:=T_Axis);
			IF fb_ConvertParaAxis.xDone OR fb_ConvertParaAxis.xError THEN
				IF (T_Axis.T_Config_Setting.rHCRampDeceleration = 0) THEN T_Axis.T_Config_Setting.rHCRampDeceleration:=20000.0; END_IF;
				IF (T_Axis.T_Config_Setting.rHCRampJerk = 0) THEN T_Axis.T_Config_Setting.rHCRampJerk:=7000.0; END_IF;
				IF fb_ConvertParaAxis.xError THEN
					fb_ConvertParaAxis(	xStart:=FALSE,
										T_Axis:=T_Axis);
					(* active step error *)
					iStepFile:=94;
				ELSE
					(* activ state read successfull *)
					iStepFile:=98;
				END_IF;
			END_IF;
		(* start time out *)
		11:	TimerFileLocked(IN:=FALSE);
			(* next step *)
			iStepFile:=iStepFile+1;
		(* prepare data *)
		12:	(* copy data *)
			i:=1;
			WHILE T_Axis.T_FileObj.sData[i] <> '' AND i <= csiMaxAxisFileObj AND i <= csiMaxFileLine DO
				T_HDD.T_Data.sData[i]:=T_Axis.T_FileObj.sData[i];
				(* next line *)
				i:=i+1;
			END_WHILE
			(* next step *)
			iStepFile:=iStepFile+1;
		(* start write file *)
		13:	IF T_HDD.T_Ctrle.xDone  AND NOT(T_HDD.T_Ctrle.xLocked) THEN
			(* activ write axis parameter *)
				T_HDD.T_Ctrle.xExecute:=TRUE;
				T_HDD.T_Ctrle.xLocked :=TRUE;
				T_HDD.T_Ctrle.iFunction:=3;
				sTmp:=CONCAT(cssRootPLC,'\Hard Disk\Bore800\Axis\File\');
				sTmp:=CONCAT(sTmp, T_Axis.T_Config_Gen.sDeviceFileName);
				T_HDD.T_File.sPathAndFileName:=CONCAT(sTmp,'.txt');
				(* next step *)
				iStepFile:=iStepFile+1;
			ELSE
			(* activ error if time out done, HDD not ready *)
				IF TimerFileLocked.Q THEN
					iStepFile:=92;
				END_IF
			END_IF
		(* wait done or error *)
		14:	IF T_HDD.T_Ctrle.xDone OR T_HDD.T_Ctrle.xErr THEN
				IF T_HDD.T_Ctrle.xErr  THEN
				(* active step error *)
					iStepFile:=93;
				ELSE
				(* activ state write successfull *)
					iStepFile:=98;
				END_IF
			END_IF
		(* start read error *)
		91:	T_Axis.T_CtrleSingle.xDone:=FALSE;
			T_Axis.T_CtrleSingle.udiErrorID:=16#F104;
			(* last step *)
			iStepFile:=99;
		(* start write error *)
		92:	T_Axis.T_CtrleSingle.xDone:=FALSE;
			T_Axis.T_CtrleSingle.udiErrorID:=16#F105;
			(* last step *)
			iStepFile:=99;
		(* block function error *)
		93:	T_Axis.T_CtrleSingle.xDone:=FALSE;
			T_Axis.T_CtrleSingle.udiErrorID:=T_HDD.T_Ctrle.udiErrorID;
			(* last step *)
			iStepFile:=99;
		(* Config File Error *)
		94:	T_Axis.T_CtrleSingle.xDone:=FALSE;
			T_Axis.T_CtrleSingle.udiErrorID:=16#F202;
			(* last step *)
			iStepFile:=99;
		(* init. successfully ended *)
		98:	T_Axis.T_CtrleSingle.xDone:=TRUE;
			T_Axis.T_CtrleSingle.xErr:= FALSE;
			T_Axis.T_CtrleSingle.udiErrorID:=16#0;
			(* last step *)
			iStepFile:=99;
		(* init. done *)
		99:	IF T_HDD.T_Ctrle.xErr AND NOT(T_HDD.T_Ctrle.xReset)THEN
				IF (T_Axis.T_CtrleSingle.udiErrorID = 1804) THEN
					T_Axis.T_CtrleSingle.udiErrorID:=16#F201;		(* File not Found *)
				END_IF;
				T_HDD.T_Ctrle.xReset:=TRUE;
				RETURN;
			END_IF;
			IF NOT(T_HDD.T_Ctrle.xDone) THEN
				RETURN;
			END_IF;
			IF NOT(T_Axis.T_CtrleSingle.xDone) THEN
				T_Axis.T_CtrleSingle.xErr:= TRUE;
			END_IF;
			xReadFile:=FALSE;
			xWriteFile:=FALSE;
			T_HDD.T_Ctrle.xExecute:=FALSE;
			(* locked off *)
			T_HDD.T_Ctrle.xLocked:=FALSE;
		ELSE
;
		END_CASE
	END_IF

(* Power function *)
	RisingEdgePowerOn(CLK:=xPowerOn);
	RisingEdgePowerOff(CLK:=xPowerOff);
	IF xPowerOn THEN
		fbAxisPower(	Enable:=TRUE,
					Enable_Positive:=TRUE,
					Enable_Negative:=TRUE,
					AxisRefIn:=T_AxisRefIn,
					AxisRefOut:=T_AxisRefOut);
		T_Axis.T_CtrleSingle.xPower:=fbAxisPower.Status;
		(* desactiv control flag during sending axis parameter and during reset  *)
		IF NOT(xSendAxisParameter) AND NOT(xResetAxis) THEN
			IF RisingEdgePowerOn.Q AND  NOT(fbAxisPower.Error) THEN
				T_Axis.T_CtrleSingle.xDone:=TRUE;
			END_IF
			IF  fbAxisPower.Error THEN
				T_Axis.T_CtrleSingle.xErr:= fbAxisPower.Error;
				T_Axis.T_CtrleSingle.udiErrorID:=fbAxisPower.ErrorID;
			END_IF
		END_IF
	END_IF
	IF xPowerOff THEN
		fbAxisPower(	Enable:=FALSE,
					AxisRefIn:=T_AxisRefIn,
					AxisRefOut:=T_AxisRefOut);
		T_Axis.T_CtrleSingle.xPower:=fbAxisPower.Status;
		(* desactiv control flag during sending axis parameter and during reset *)
		IF NOT(xSendAxisParameter) AND NOT(xResetAxis) THEN
			IF RisingEdgePowerOff.Q AND NOT( fbAxisPower.Error) THEN
				T_Axis.T_CtrleSingle.xDone:=TRUE;
			END_IF
			IF  fbAxisPower.Error THEN
				T_Axis.T_CtrleSingle.xErr:= fbAxisPower.Error;
				T_Axis.T_CtrleSingle.udiErrorID:=fbAxisPower.ErrorID;
			END_IF
		END_IF
	END_IF

(* Stop *)
	IF xStop THEN
		(* init. FB vel / abs / rel *)
		xMoveVel:=FALSE;
		xMoveRel:=FALSE;
		xMoveAbs:=FALSE;
		xMoveModulo:=FALSE;
		xNewVelocity:=FALSE;
		xNewPosition:=FALSE;
		xStartTimerComm:=FALSE;
		xHoming:=FALSE;
		IF (iTmpFctNr <> 19) THEN
			xCalcAngleRefIndex:=FALSE;
		END_IF;
		(* flag oscillation off *)
		xOscillation:=FALSE;
		(* FB stop *)
		fbAxisStop(	Execute:=TRUE,
					Deceleration:=T_Axis.T_CtrleSingle.lrDecceleration,
					Jerk:=T_Axis.T_CtrleSingle.lrJerk,
					Axis:=T_AxisRefIn);
		(* select bit not moving *)
		dwTmp:=T_Axis.T_LiveValue.dwState AND 16#4;
		IF (fbAxisStop.Done AND dwTmp = 16#4) OR fbAxisStop.Error THEN
			IF fbAxisStop.Error OR (NOT(xResetAxis) AND NOT(xCalcAngleRefIndex) )THEN
				xResetAxis:=xCalcAngleRefIndex:=FALSE;
			(* confirm reset if error activ or if reset is not activ *)
				T_Axis.T_CtrleSingle.xDone:=fbAxisStop.Done;
				T_Axis.T_CtrleSingle.xErr:= fbAxisStop.Error;
				T_Axis.T_CtrleSingle.udiErrorID:=fbAxisStop.ErrorID;
				(* desactiv reset axis *)
				IF xResetAxis THEN xResetAxis:=FALSE; END_IF
			END_IF
			(* flag stop off *)
			xStop:=FALSE;
			tTimeCommLeft1:=TimerCommTimeLeft1.ET;
			xStartTimerComm1:=FALSE;
			(* reset flag busy *)
			T_Axis.T_CtrleSingle.xBusyNewPosAndVel:=FALSE;
			(* Init. Stop FB *)
			fbAxisStop(Execute:=FALSE, Axis:=T_AxisRefIn);
		END_IF
	ELSE fbAxisStop(Execute:=FALSE, Axis:=T_AxisRefIn); END_IF

(* Velocity *)
	IF xMoveVel AND NOT(fbAxisMoveVelocity.InVelocity) THEN
		IF T_Axis.T_CtrleSingle.lrVelocity >= 0 THEN
		(* positiv direction =1*)
			iDirectionVel:=MC_Positive_Direction;
		ELSE
		(* negativ direction =3*)
			iDirectionVel:=MC_Negative_Direction;
		END_IF
		rVelocity:=ABS(lrOverrideVel);
		fbAxisMoveVelocity(	Execute:=TRUE,
							Velocity:=rVelocity,
							Acceleration:=T_Axis.T_CtrleSingle.lrAcceleration,
							Deceleration:=T_Axis.T_CtrleSingle.lrDecceleration,
							Jerk:=T_Axis.T_CtrleSingle.lrJerk,
							Direction:=iDirectionVel,
							Axis:=T_AxisRefIn);
		IF fbAxisMoveVelocity.InVelocity OR fbAxisMoveVelocity.Error THEN
			T_Axis.T_CtrleSingle.xDone:=fbAxisMoveVelocity.InVelocity;
			T_Axis.T_CtrleSingle.xErr:= fbAxisMoveVelocity.Error;
			T_Axis.T_CtrleSingle.udiErrorID:=fbAxisMoveVelocity.ErrorID;
			(* flag velocity off *)
			xMoveVel:=FALSE;
			(* Init. FB Move *)
			fbAxisMoveVelocity(Execute:=FALSE, Axis:=T_AxisRefIn);
		END_IF
	ELSE fbAxisMoveVelocity(Execute:=FALSE, Axis:=T_AxisRefIn); END_IF

(* Move absolute *)
	IF xMoveAbs THEN
		fbAxisMoveAbsolute(	Execute:=TRUE,
							Position:=T_Axis.T_CtrleSingle.lrPosition,
							Velocity:=ABS(lrOverrideVel),
							Acceleration:=T_Axis.T_CtrleSingle.lrAcceleration,
							Deceleration:=T_Axis.T_CtrleSingle.lrDecceleration,
							Jerk:=T_Axis.T_CtrleSingle.lrJerk,
							Axis:=T_AxisRefIn);
		IF fbAxisMoveAbsolute.Done OR fbAxisMoveAbsolute.Error THEN
			IF NOT(xCalcAngleRefIndex) OR fbAxisMoveAbsolute.Error THEN
				xCalcAngleRefIndex:=FALSE;
				T_Axis.T_CtrleSingle.xDone:=fbAxisMoveAbsolute.Done;
				T_Axis.T_CtrleSingle.xErr:= fbAxisMoveAbsolute.Error;
				T_Axis.T_CtrleSingle.udiErrorID:=fbAxisMoveAbsolute.ErrorID;
				(* test if move has been stopped *)
				IF fbAxisMoveAbsolute.ErrorID = 16#4B00 THEN
				(* clear error *)
					T_Axis.T_CtrleSingle.xDone:=TRUE;
					T_Axis.T_CtrleSingle.xErr:= FALSE;
					T_Axis.T_CtrleSingle.udiErrorID:=16#0;
				END_IF
			END_IF;
			(* flag move absolute off *)
			xMoveAbs:=FALSE;
			(* init. FB *)
			fbAxisMoveAbsolute(Execute:=FALSE, Axis:=T_AxisRefIn);
		END_IF
	ELSE fbAxisMoveAbsolute(Execute:=FALSE, Axis:=T_AxisRefIn); END_IF

(* Move relative *)
	IF xMoveRel THEN
		fbAxisMoveRelative(	Execute:=TRUE,
							Distance:=T_Axis.T_CtrleSingle.lrDistance,
							Velocity:=lrOverrideVel,
							Acceleration:=T_Axis.T_CtrleSingle.lrAcceleration,
							Deceleration:=T_Axis.T_CtrleSingle.lrDecceleration,
							Jerk:=T_Axis.T_CtrleSingle.lrJerk,
							Axis:=T_AxisRefIn);
		IF fbAxisMoveRelative.Done OR fbAxisMoveRelative.Error THEN
			IF (NOT(xOscillation) AND NOT(xCalcAngleRefIndex)) OR fbAxisMoveRelative.Error THEN
				xOscillation:=xCalcAngleRefIndex:=FALSE;
			(* normal control variable settings if oscillation disable *)
				T_Axis.T_CtrleSingle.xDone:=fbAxisMoveRelative.Done;
				T_Axis.T_CtrleSingle.xErr:= fbAxisMoveRelative.Error;
				T_Axis.T_CtrleSingle.udiErrorID:=fbAxisMoveRelative.ErrorID;
				(* test if move has been stopped *)
				IF fbAxisMoveRelative.ErrorID = 16#4B00 THEN
				(* clear error *)
					T_Axis.T_CtrleSingle.xDone:=TRUE;
					T_Axis.T_CtrleSingle.xErr:= FALSE;
					T_Axis.T_CtrleSingle.udiErrorID:=16#0;
				END_IF
			END_IF
			(* flag move relative off *)
			xMoveRel:=FALSE;
			(* init. FB *)
			fbAxisMoveRelative(Execute:=FALSE, Axis:=T_AxisRefIn);
		END_IF
	ELSE fbAxisMoveRelative(Execute:=FALSE, Axis:=T_AxisRefIn); END_IF

(* Move modulo *)
	IF xMoveModulo THEN
		fbAxisMoveModulo(	Execute:= TRUE,
							Position:= T_Axis.T_CtrleSingle.lrPosition,
							Velocity:= ABS(lrOverrideVel),
							Acceleration:= T_Axis.T_CtrleSingle.lrAcceleration,
							Deceleration:= T_Axis.T_CtrleSingle.lrDecceleration,
							Jerk:= T_Axis.T_CtrleSingle.lrJerk,
							Direction:= T_Axis.T_CtrleSingle.iModuloDirection,
							Axis:= T_AxisRefIn);
		IF fbAxisMoveModulo.Done OR fbAxisMoveModulo.Error THEN
			xCalcAngleRefIndex:=FALSE;
			T_Axis.T_CtrleSingle.xDone:=fbAxisMoveModulo.Done;
			T_Axis.T_CtrleSingle.xErr:= fbAxisMoveModulo.Error;
			T_Axis.T_CtrleSingle.udiErrorID:=fbAxisMoveModulo.ErrorID;
			(* test if move has been stopped *)
			IF fbAxisMoveModulo.ErrorID = 16#4B00 THEN
			(* clear error *)
				T_Axis.T_CtrleSingle.xDone:=TRUE;
				T_Axis.T_CtrleSingle.xErr:= FALSE;
				T_Axis.T_CtrleSingle.udiErrorID:=16#0;
			END_IF
			(* flag move absolute off *)
			xMoveModulo:=FALSE;
			(* init. FB *)
			fbAxisMoveModulo(Execute:=FALSE, Axis:=T_AxisRefIn);
		END_IF
	ELSE fbAxisMoveModulo(Execute:=FALSE, Axis:=T_AxisRefIn); END_IF

(* Homing *)
	IF xHoming THEN
		fbAxisHoming(	Execute:=TRUE,
						Position:=T_Axis.T_CtrleSingle.rSetPosition,
						bCalibrationCam:=xRefHoming,
						Axis:=T_AxisRefIn,
						AxisOut:=T_AxisRefOut);
		IF fbAxisHoming.Done OR fbAxisHoming.Error THEN
			IF NOT(xCalcAngleRefIndex) OR fbAxisHoming.Error THEN
				xCalcAngleRefIndex:=FALSE;
				T_Axis.T_CtrleSingle.xDone:=fbAxisHoming.Done;
				T_Axis.T_CtrleSingle.xErr:= fbAxisHoming.Error;
				T_Axis.T_CtrleSingle.udiErrorID:=fbAxisHoming.ErrorID;
			END_IF;
			(* flag homing off *)
			xHoming:=FALSE;
			(* Init. FB Homing *)
			fbAxisHoming(	Execute:=FALSE,
							Axis:=T_AxisRefIn,
							AxisOut:=T_AxisRefOut);
		END_IF
	ELSE
		fbAxisHoming(	Execute:=FALSE,
						Axis:=T_AxisRefIn,
						AxisOut:=T_AxisRefOut);
	END_IF

(* Set override *)
	IF xOverride THEN
		fbAxisSetOverride(Execute:=TRUE,
						Override:=T_Axis.T_CtrleSingle.dwOverride,
						AxisRefIn:=T_AxisRefIn,
						AxisRefOut:=T_AxisRefOut);
		IF fbAxisSetOverride.Done OR fbAxisSetOverride.Error THEN
			T_Axis.T_CtrleSingle.xDone:=fbAxisSetOverride.Done;
			T_Axis.T_CtrleSingle.xErr:= fbAxisSetOverride.Error;
			T_Axis.T_CtrleSingle.udiErrorID:=fbAxisSetOverride.ErrorID;
			(* flag override off *)
			xOverride:=FALSE;
			(* Init. FB Override *)
			fbAxisSetOverride(Execute:=FALSE,
							AxisRefIn:=T_AxisRefIn,
							AxisRefOut:=T_AxisRefOut);
		END_IF
	ELSE
		fbAxisSetOverride(Execute:=FALSE,
						AxisRefIn:=T_AxisRefIn,
						AxisRefOut:=T_AxisRefOut);
	END_IF

(* Set new position *)
	IF xSetPosition THEN
		fbAxisSetPosition(	Execute:=TRUE, Position:=T_Axis.T_CtrleSingle.rSetPosition, Axis:=T_AxisRefIn);
		IF fbAxisSetPosition.Done OR fbAxisSetPosition.Error THEN
			T_Axis.T_CtrleSingle.xDone:=fbAxisSetPosition.Done;
			T_Axis.T_CtrleSingle.xErr:= fbAxisSetPosition.Error;
			T_Axis.T_CtrleSingle.udiErrorID:=fbAxisSetPosition.ErrorID;
			(* flag set position off *)
			xSetPosition:=FALSE;
			(* Init. FB set position *)
			fbAxisSetPosition(Execute:=FALSE, Axis:=T_AxisRefIn);
		END_IF
	ELSE fbAxisSetPosition(Execute:=FALSE, Axis:=T_AxisRefIn); END_IF

(* set new velocity or new position *)
	IF xNewVelocity OR xNewPosition THEN
		IF NOT(xOscillation) OR xNewPosition THEN
			IF NOT(T_Axis.T_CtrleSingle.xNotMoving) THEN
				xNoHWError:=FALSE;
				IF xNewVelocity THEN
				(* new velocity *)
					fbAxisNewPosAndVel(	Execute:=TRUE,
										Mode:=2,
										NewVelo:=ABS(lrOverrideVel),
										Axis:=T_AxisRefIn);
				ELSE
				(* new position *)
					fbAxisNewPosAndVel(	Execute:=TRUE,
										Mode:=3,
										NewPos:=T_Axis.T_CtrleSingle.lrPosition,
										NewVelo:=lrOverrideVel,
										Axis:=T_AxisRefIn);
				END_IF
			ELSE
				xNoHWError:=TRUE;
			END_IF;
			IF fbAxisNewPosAndVel.Done OR fbAxisNewPosAndVel.Error OR xNoHWError THEN
			(* confirm end function *)
				IF xMovement THEN
					IF NOT(xNoHWError) THEN
						T_Axis.T_CtrleSingle.xDone:=FALSE;
					ELSE
						IF xMoveAbs OR xMoveRel OR xMoveModulo THEN
							T_Axis.T_CtrleSingle.xDone:=FALSE;
						ELSE
							T_Axis.T_CtrleSingle.xDone:=TRUE;
						END_IF;
					END_IF;
				ELSE
					IF NOT(xNoHWError) THEN
						T_Axis.T_CtrleSingle.xDone:=fbAxisNewPosAndVel.Done;
					ELSE
						T_Axis.T_CtrleSingle.xDone:=TRUE;
					END_IF;
				END_IF;
				IF NOT(xNoHWError) THEN
					T_Axis.T_CtrleSingle.xErr:= fbAxisNewPosAndVel.Error;
					T_Axis.T_CtrleSingle.udiErrorID:=fbAxisNewPosAndVel.ErrorID;
				ELSE
					xNoHWError:=FALSE;
					T_Axis.T_CtrleSingle.xErr:= FALSE;
					T_Axis.T_CtrleSingle.udiErrorID:=0;
				END_IF;
				(* flag new velocity off and new position off *)
				xNewVelocity:=FALSE;
				xNewPosition:=FALSE;
				T_Axis.T_CtrleSingle.iFunction:=iTmpFctNr;
				(* Init. flag busy *)
				T_Axis.T_CtrleSingle.xBusyNewPosAndVel:=FALSE;
				(* Init. FB New pos and vel *)
				fbAxisNewPosAndVel(	Execute:=FALSE, Axis:=T_AxisRefIn);
				tTimeCommLeft:=TimerCommTimeLeft.ET;
				xStartTimerComm:=FALSE;
			END_IF
		ELSE
			(* velocity calculation *)
			IF T_Axis.T_Oscillation.rFrequence >= 0 AND T_Axis.T_Oscillation.rFrequence <= 1 THEN
				rTmpFrequence:=1.05 * T_Axis.T_Oscillation.rFrequence; END_IF
			IF T_Axis.T_Oscillation.rFrequence >=1 AND T_Axis.T_Oscillation.rFrequence <= 2 THEN
				rTmpFrequence:=1.25 * T_Axis.T_Oscillation.rFrequence; END_IF
			IF T_Axis.T_Oscillation.rFrequence >= 2 AND T_Axis.T_Oscillation.rFrequence <= 3 THEN
				rTmpFrequence:=2.5 * T_Axis.T_Oscillation.rFrequence; END_IF
			IF T_Axis.T_Oscillation.rFrequence >= 3 AND T_Axis.T_Oscillation.rFrequence <= 4 THEN
				rTmpFrequence:=5 * T_Axis.T_Oscillation.rFrequence; END_IF
			IF T_Axis.T_Oscillation.rFrequence >= 4 AND T_Axis.T_Oscillation.rFrequence <= 5 THEN
				rTmpFrequence:=10 * T_Axis.T_Oscillation.rFrequence; END_IF
			IF T_Axis.T_Oscillation.rFrequence > 5 THEN rTmpFrequence:=20; END_IF
			lrTmpVelocity:=(rTmpFrequence * 2 + 1 / rTmpFrequence) * ABS(T_Axis.T_Oscillation.rOffset);
			IF lrTmpVelocity > 250 THEN T_Axis.T_CtrleSingle.lrVelocity:=250;
				ELSE T_Axis.T_CtrleSingle.lrVelocity:=lrTmpVelocity; END_IF
			IF xMovement THEN
				T_Axis.T_CtrleSingle.xDone:=FALSE;
			ELSE
				T_Axis.T_CtrleSingle.xDone:=TRUE;
			END_IF;
			T_Axis.T_CtrleSingle.xErr:= FALSE;
			T_Axis.T_CtrleSingle.udiErrorID:=0;
			xNewVelocity:=FALSE;
			T_Axis.T_CtrleSingle.iFunction:=iTmpFctNr;
			T_Axis.T_CtrleSingle.xBusyNewPosAndVel:=FALSE;
			tTimeCommLeft:=TimerCommTimeLeft.ET;
			xStartTimerComm:=FALSE;
		END_IF;
	ELSE IF NOT(xNewVelocity) AND NOT( xNewPosition) THEN fbAxisNewPosAndVel(Execute:=FALSE, Axis:=T_AxisRefIn); END_IF
	END_IF

(* Set or reset reference flag *)
	IF xSetReferenceFlag OR xResetReferenceFlag THEN
		IF xSetReferenceFlag THEN
		(* set reference flag *)
			xTmp:=TRUE;
		ELSE xTmp:=FALSE;
		END_IF
		fbAxisSetReferenceFlag(Execute:=TRUE, ReferenceFlag:=xTmp, Axis:=T_AxisRefIn);
		IF fbAxisSetReferenceFlag.Done OR fbAxisSetReferenceFlag.Error THEN
			T_Axis.T_CtrleSingle.xDone:=fbAxisSetReferenceFlag.Done;
			T_Axis.T_CtrleSingle.xErr:= fbAxisSetReferenceFlag.Error;
			T_Axis.T_CtrleSingle.udiErrorID:=fbAxisSetReferenceFlag.ErrorID;
			(* set flag 'reference flag' off *)
			xSetReferenceFlag:=FALSE;
			xResetReferenceFlag:=FALSE;
			(* Init. FB set reference *)
			fbAxisSetReferenceFlag(Execute:=FALSE, Axis:=T_AxisRefIn);
		END_IF
	ELSE fbAxisSetReferenceFlag(Execute:=FALSE, Axis:=T_AxisRefIn); END_IF

(* set/reset control position *)
	IF xCtrlePositionOn THEN
		fbExtSetPointGenEnable(	Execute:=TRUE,
								Axis:=T_AxisRefIn);
		IF fbExtSetPointGenEnable.Done OR fbExtSetPointGenEnable.Error THEN
			T_Axis.T_CtrleSingle.xDone:=fbExtSetPointGenEnable.Done;
			T_Axis.T_CtrleSingle.xErr:= fbExtSetPointGenEnable.Error;
			T_Axis.T_CtrleSingle.udiErrorID:=fbExtSetPointGenEnable.ErrorID;
			(* reset flag *)
			xCtrlePositionOn:=FALSE;
		END_IF
	ELSE
		fbExtSetPointGenEnable(	Execute:=FALSE,
								Axis:=T_AxisRefIn);
	END_IF
	IF xCtrlePositionOff THEN
		fbExtSetPointGenDisable(	Execute:=TRUE,
								Axis:=T_AxisRefIn);
		IF fbExtSetPointGenDisable.Done OR fbExtSetPointGenDisable.Error THEN
			T_Axis.T_CtrleSingle.xDone:=fbExtSetPointGenDisable.Done;
			T_Axis.T_CtrleSingle.xErr:= fbExtSetPointGenDisable.Error;
			T_Axis.T_CtrleSingle.udiErrorID:=fbExtSetPointGenDisable.ErrorID;
			(* reset flag *)
			xCtrlePositionOff:=FALSE;
		END_IF
	ELSE
		fbExtSetPointGenDisable(	Execute:=FALSE,
								Axis:=T_AxisRefIn);
	END_IF

(* calcultate angle between Reference Index and Reference Sensor *)
	IF xCalcAngleRefIndex THEN
		(* error or stop => stop oscillation *)
		IF T_Axis.T_CtrleSingle.xErr OR (xStop AND (iTmpFctNr <> 19)) THEN iStepOsc:=99; END_IF
		CASE iStepCalcRefIndex OF
		(* Drive referencing and search the Ref. Index *)
		1:	T_Axis.T_CtrleSingle.rSetPosition:=0.0;
			xHoming:=TRUE;
			iStepCalcRefIndex:=10;
			T_Axis.T_CtrleSingle.iStrokeAngleRefIndex:=0;
			lrTechUnitPerMotorTurn:=65536.0 * T_Axis.T_Config_ObjFileValue.lrScaleFactor;	(*65536 = inc pro Motorumdrehung-->so kann dann mit dem Skalierungsfaktor ermittelt werden, wieviel Tech.Einheit für eine Motorumdrehung*)
			IF lrTechUnitPerMotorTurn = 0.0 THEN
				IF (T_Axis.T_Config_Gen.iTyp = 1) THEN
					lrTechUnitPerMotorTurn:=2.5;	(* 2.5mm entsprechen einer Motorumdrehung *)
				END_IF;
				IF (T_Axis.T_Config_Gen.iTyp = 4) THEN
					lrTechUnitPerMotorTurn:=30.0;	(* 30 Grad entsprechen einer Motorumdrehung *)
				END_IF;
			END_IF;
		10:	IF NOT(xHoming) THEN
				(* Go Absolut to the Reference Index *)
				T_Axis.T_CtrleSingle.lrPosition:=0.0;
				T_Axis.T_CtrleSingle.lrVelocity:=1.0;(*T_Axis.T_Config_ObjFileValue.lrCalVelocityBackward;*)
				T_Axis.T_CtrleSingle.lrAcceleration:=T_Axis.T_Config_ObjFileValue.lrAcceleration;
				T_Axis.T_CtrleSingle.lrDecceleration:=T_Axis.T_Config_ObjFileValue.lrDecceleration;
				T_Axis.T_CtrleSingle.lrJerk:=T_Axis.T_Config_ObjFileValue.lrJerk;
				xMoveAbs:=TRUE;
				iStepCalcRefIndex:=20;
			END_IF;
		20:	IF NOT(xMoveAbs) THEN
				(* Turn the Motor for 360 degrees relativ*)
				xCheckRefState:=xRefHoming;
				T_Axis.T_CtrleSingle.lrDistance:=lrTechUnitPerMotorTurn * -1.0;	(* Der eingesetzte Wert entscheidet ob links oder rechtsdrehend, daher ist es wichtig zu wissen dass der entsprechende Wert, Positiv oder Negativ, die Bewegung zum Ref.Sensor führt *)
				T_Axis.T_CtrleSingle.lrVelocity:=1.0;(*T_Axis.T_Config_ObjFileValue.lrCalVelocityBackward;*)
				T_Axis.T_CtrleSingle.lrAcceleration:=T_Axis.T_Config_ObjFileValue.lrAcceleration;
				T_Axis.T_CtrleSingle.lrDecceleration:=T_Axis.T_Config_ObjFileValue.lrDecceleration;
				T_Axis.T_CtrleSingle.lrJerk:=T_Axis.T_Config_ObjFileValue.lrJerk;
				xMoveRel:=TRUE;
				iStepCalcRefIndex:=30;
			END_IF;
		30:	T_Axis.T_CtrleSingle.iStrokeAngleRefIndex:=ABS(LREAL_TO_INT((360.0 / lrTechUnitPerMotorTurn) * T_Axis.T_LiveValue.lrActualPosition));	(* Zeiger bewegt sich so dynamisch während der Fahrt auf der Suche des RefSensors *)
			IF xCheckRefState XOR xRefHoming THEN
				lrCapturePosition:=T_Axis.T_LiveValue.lrActualPosition;
				IF (ABS(lrCapturePosition) > ABS(lrTechUnitPerMotorTurn)) THEN
					lrCapturePosition:=360.0 - ABS(lrCapturePosition);
				END_IF;
				xStop:=TRUE;
				iStepCalcRefIndex:=40;
			END_IF;
			IF NOT(xMoveRel) AND NOT(xStop) THEN
				T_Axis.T_CtrleSingle.iStrokeAngleRefIndex:=0;
				iStepCalcRefIndex:=50;
			END_IF;
		40:	IF NOT(xStop) THEN
				T_Axis.T_CtrleSingle.iStrokeAngleRefIndex:=LREAL_TO_INT((360.0 / lrTechUnitPerMotorTurn) * lrCapturePosition);	(* Berechnung der Winkellage des RefIndex zum RefSensor *)
				IF (T_Axis.T_CtrleSingle.iStrokeAngleRefIndex < 0) THEN
					T_Axis.T_CtrleSingle.iStrokeAngleRefIndex:=T_Axis.T_CtrleSingle.iStrokeAngleRefIndex * -1;
				END_IF;
				IF (T_Axis.T_CtrleSingle.iStrokeAngleRefIndex > 360) THEN
					T_Axis.T_CtrleSingle.iStrokeAngleRefIndex:=360;
				END_IF;
				iStepCalcRefIndex:=50;
			END_IF;
		(* End of calc of the ref index position *)
		50:	T_Axis.T_CtrleSingle.xDone:=TRUE;
			T_Axis.T_CtrleSingle.xErr:= FALSE;
			T_Axis.T_CtrleSingle.udiErrorID:=16#0;
			xCalcAngleRefIndex:=FALSE;
		END_CASE;
	ELSE
		iStepCalcRefIndex:=1;
	END_IF;

(* Oscillation *)
	IF xOscillation THEN
		(* error or stop => stop oscillation *)
		IF T_Axis.T_CtrleSingle.xErr OR xStop THEN iStepOsc:=99; END_IF
		CASE iStepOsc OF
		(* init. oscillation + start move*)
		1:	(* init. variable *)
			iOscCounter:=0;
			(* velocity calculation *)
			IF T_Axis.T_Oscillation.rFrequence >= 0 AND T_Axis.T_Oscillation.rFrequence <= 1 THEN
				rTmpFrequence:=1.05 * T_Axis.T_Oscillation.rFrequence; END_IF
			IF T_Axis.T_Oscillation.rFrequence >=1 AND T_Axis.T_Oscillation.rFrequence <= 2 THEN
				rTmpFrequence:=1.25 * T_Axis.T_Oscillation.rFrequence; END_IF
			IF T_Axis.T_Oscillation.rFrequence >= 2 AND T_Axis.T_Oscillation.rFrequence <= 3 THEN
				rTmpFrequence:=2.5 * T_Axis.T_Oscillation.rFrequence; END_IF
			IF T_Axis.T_Oscillation.rFrequence >= 3 AND T_Axis.T_Oscillation.rFrequence <= 4 THEN
				rTmpFrequence:=5 * T_Axis.T_Oscillation.rFrequence; END_IF
			IF T_Axis.T_Oscillation.rFrequence >= 4 AND T_Axis.T_Oscillation.rFrequence <= 5 THEN
				rTmpFrequence:=10 * T_Axis.T_Oscillation.rFrequence; END_IF
			IF T_Axis.T_Oscillation.rFrequence > 5 THEN rTmpFrequence:=20; END_IF
			lrTmpVelocity:=(rTmpFrequence * 2 + 1 / rTmpFrequence) * ABS(T_Axis.T_Oscillation.rOffset);
			IF lrTmpVelocity > 250 THEN T_Axis.T_CtrleSingle.lrVelocity:=250;
				ELSE T_Axis.T_CtrleSingle.lrVelocity:=lrTmpVelocity; END_IF
			(*
			(* velocity := frequence * (offset * 2) *)
			T_Axis.T_CtrleSingle.lrVelocity:=T_Axis.T_Oscillation.rFrequence * ABS(T_Axis.T_Oscillation.rOffset) * 2;
			*)
			(* set move *)
			T_Axis.T_CtrleSingle.lrDistance:=T_Axis.T_Oscillation.rOffset;
			xMoveRel:=TRUE;
			(* next step *)
			iStepOsc:=10;
		(* move *)
		10:	IF NOT(xMoveRel) THEN
				(* move *-1 *)
				T_Axis.T_CtrleSingle.lrDistance:=T_Axis.T_Oscillation.rOffset * -1;
				xMoveRel:=TRUE;
				(* next step *)
				iStepOsc:=20;
			END_IF
		(* osc +1 *)
		20:	IF NOT(xMoveRel) THEN
				iOscCounter:=iOscCounter+1;
				IF iOscCounter < T_Axis.T_Oscillation.iCycle THEN
				(* move *)
					T_Axis.T_CtrleSingle.lrDistance:=T_Axis.T_Oscillation.rOffset;
					xMoveRel:=TRUE;
					(* next step *)
					iStepOsc:=10;
				ELSE
				(* oscillation done *)
					T_Axis.T_CtrleSingle.xDone:=TRUE;
					T_Axis.T_CtrleSingle.xErr:= FALSE;
					T_Axis.T_CtrleSingle.udiErrorID:=16#0;
					(* init FB *)
					fbAxisMoveRelative(Execute:=FALSE, Axis:=T_AxisRefIn);
					(* reset flag *)
					xOscillation:=FALSE;
				END_IF
			END_IF
		(* end oscillation *)
		99:	xOscillation:=FALSE;
		END_CASE
	ELSE
	(* init. variable *)
		iStepOsc:=1;
	END_IF

(* Default parameter value *)
	IF xDefaultAxisParameter THEN
		fbDefaultAxisPara(xDefaultValue:=TRUE,T_Axis:=T_Axis);
		T_Axis.T_CtrleSingle.xDone:=TRUE;
		T_Axis.T_CtrleSingle.xErr:= FALSE;
		T_Axis.T_CtrleSingle.udiErrorID:=0;
		(* flag DefaultParameter off *)
		xDefaultAxisParameter:=FALSE;
	END_IF

(* Send parameter *)
	IF xSendAxisParameter THEN
		CASE iStepSendPara OF
		(* control flag *)
		1:	(* init. next step *)
			iStepSendPara:=2;
			IF T_Axis.T_CtrleSingle.xPower THEN
			(* axis power on, control axis flag *)
				IF (T_AxisRefIn.nStateDWord AND 16#4) = 16#0 THEN
				(* axis is moving, activ error *)
					iStepSendPara:=912;
				END_IF
				IF (T_AxisRefIn.nStateDWord AND 16#20) = 16#20 THEN
				(* axis is in slave mode, activ error *)
					iStepSendPara:=913;
				END_IF
			END_IF
		(* set power off *)
		2:	xRestoreAxisPower:=FALSE;
			IF T_Axis.T_CtrleSingle.xPower THEN
			(* set power off *)
				xPowerOff:=TRUE;
				xPowerOn:=NOT(xPowerOff);
				(* set flag restore *)
				xRestoreAxisPower:=TRUE;
				(* start time out *)
				TimerOutSendPara(IN:=FALSE);
				(* next step *)
				iStepSendPara:=3;
			ELSE
			(* already power off, activ send parameter *)
				iStepSendPara:=11;
			END_IF
		(* wait flag power off *)
		3:	IF NOT(T_Axis.T_CtrleSingle.xPower) THEN
			(* activ send parameter *)
				iStepSendPara:=11;
				xSendBlock:=FALSE;
			END_IF
			IF TimerOutSendPara.Q THEN
			(* time out activ, set error *)
				iStepSendPara:=911;
			END_IF
		(* loop sending parameter *)
		11:	IF NOT (fbAdsWrite.BUSY )  AND NOT(xSendBlock) THEN
			(* send axis parameter *)
				fbAdsWrite(WRITE:=FALSE);
				CASE T_Axis.T_ParamFileObj[iPtrAxisParameter].udiLength OF
				(* True/False, 2 bytes*)
				2:	wTmp:=LREAL_TO_WORD(T_Axis.T_ParamFileObj[iPtrAxisParameter].lrReal);
					dwAdrVar:=ADR(wTmp);
				(* dword value, 4 bytes *)
				4:	dwTmp:=LREAL_TO_DWORD(T_Axis.T_ParamFileObj[iPtrAxisParameter].lrReal);
					dwAdrVar:=ADR(dwTmp);
				(* else, 8 bytes *)
				8:	dwAdrVar:=ADR(T_Axis.T_ParamFileObj[iPtrAxisParameter].lrReal);
				END_CASE
				fbAdsWrite(	NETID:='',
							PORT:=501,
							IDXGRP:=T_Axis.T_ParamFileObj[iPtrAxisParameter].udiIdxGroup,
							IDXOFFS:=T_Axis.T_ParamFileObj[iPtrAxisParameter].udiIndexOffset,
							LEN:=T_Axis.T_ParamFileObj[iPtrAxisParameter].udiLength,
							SRCADDR:=dwAdrVar,
							WRITE:=TRUE,
							TMOUT:=T#2s);
				(* next parameter *)
				iPtrAxisParameter:=iPtrAxisParameter+1;
				IF T_Axis.T_ParamFileObj[iPtrAxisParameter].udiIdxGroup = 0 THEN
				(* parameter list empty *)
					xSendBlock:=TRUE;
				END_IF
			ELSE
				fbAdsWrite(WRITE:=FALSE);
			END_IF
			IF NOT(fbAdsWrite.BUSY) AND NOT(fbAdsWrite.ERR) AND T_Axis.T_ParamFileObj[iPtrAxisParameter].udiIdxGroup = 0 THEN
			(* determin the next step *)
				IF xRestoreAxisPower THEN
				(* Restore axis power *)
					iStepSendPara:=101;
				ELSE
				(* set flag end function *)
					iStepSendPara:=998;
				END_IF
			END_IF
			IF fbAdsWrite.ERR THEN
			(* set next step  *)
				iStepSendPara:=901;
			END_IF
		(* set power on *)
		101:	xPowerOn:=TRUE;
			xPowerOff:=NOT(xPowerOn);
			(* start time out *)
			TimerOutSendPara(IN:=FALSE);
			(*  next step *)
			iStepSendPara:=102;
		(* wait flag power on *)
		102:	IF T_Axis.T_CtrleSingle.xPower THEN
			(* set flag end function *)
				iStepSendPara:=998;
			END_IF
			IF TimerOutSendPara.Q THEN
			(* time out activ, set error *)
				iStepSendPara:=911;
			END_IF
		(* ads communication error *)
		901:	T_Axis.T_CtrleSingle.udiErrorID:=fbAdsWrite.ERRID;
			(* set next step *)
			iStepSendPara:=991;
		(* time out after setting axis power on/off *)
		911:	T_Axis.T_CtrleSingle.udiErrorID:=16#F101;
			(* set next step *)
			iStepSendPara:=991;
		(* error the axis is moving *)
		912:	T_Axis.T_CtrleSingle.udiErrorID:=16#F102;
			(* set next step *)
			iStepSendPara:=991;
		(* error the axis is in slave mode *)
		913:	T_Axis.T_CtrleSingle.udiErrorID:=16#F103;
			(* set next step *)
			iStepSendPara:=991;
		(* set flag error *)
		991:	T_Axis.T_CtrleSingle.xDone:=FALSE;
			T_Axis.T_CtrleSingle.xErr:= TRUE;
			(* set last step *)
			iStepSendPara:=999;
		(* set flag end function *)
		998:	T_Axis.T_CtrleSingle.xDone:=TRUE;
			T_Axis.T_CtrleSingle.xErr:= FALSE;
			T_Axis.T_CtrleSingle.udiErrorID:=0;
			(* set last step *)
			iStepSendPara:=999;
		(* reset variable *)
		999:	xSendAxisParameter:=FALSE;
		END_CASE
	ELSE
		fbAdsWrite(WRITE:=FALSE);
	END_IF

(* send axis string *)
	IF xSendAxisString THEN
		(*IF NOT(fbADS_ReadWriteString.BUSY)   AND sReturnAxis = '' THEN
			fbADS_ReadWriteString(WRTRD:=FALSE);*)
			(* add carriage return and line feed *)
			sSendAxis:=CONCAT(T_Axis.T_CtrleSingle.sSend, '$R$L$00');
			fbADS_ReadWriteString(	NETID:=T_Axis.T_Config_Gen.sServoNetId,
									PORT:=200,
									IDXGRP:=1,
									IDXOFFS:=1,
									WRITELEN:=LEN(sSendAxis)-1,
									READLEN:=LEN(sReturnAxis)-1,
									SRCADDR:=ADR(sSendAxis),
									DESTADDR:=ADR(sReturnAxis),
									WRTRD:=TRUE,
									TMOUT:=T#3s);
		(*ELSE
			fbADS_ReadWriteString(WRTRD:=FALSE);
		END_IF*)
		IF NOT(fbADS_ReadWriteString.BUSY) AND NOT(fbADS_ReadWriteString.ERR) AND sReturnAxis <> '' THEN
			IF sSendAxis = sReturnAxis THEN
			(* received string correct *)
				T_Axis.T_CtrleSingle.xDone:=TRUE;
				T_Axis.T_CtrleSingle.xErr:= FALSE;
				T_Axis.T_CtrleSingle.udiErrorID:=0;
			ELSE
			(* received string incorrect, active error *)
				T_Axis.T_CtrleSingle.xDone:=FALSE;
				T_Axis.T_CtrleSingle.xErr:= TRUE;
				T_Axis.T_CtrleSingle.udiErrorID:=16#F106;
			END_IF
			(* set flag xsendaxisstring off *)
			xSendAxisString:=FALSE;
		END_IF
		IF fbADS_ReadWriteString.ERR THEN
		(* set flag error *)
			T_Axis.T_CtrleSingle.xDone:=FALSE;
			T_Axis.T_CtrleSingle.xErr:= TRUE;
			T_Axis.T_CtrleSingle.udiErrorID:=fbADS_ReadWriteString.ERRID;
			(* set flag xsendaxisstring off *)
			xSendAxisString:=FALSE;
		END_IF
	ELSE
		fbADS_ReadWriteString(WRTRD:=FALSE);
	END_IF

(* save parameter NC axis to file *)
	IF xWriteFile THEN
;
	END_IF
END_FUNCTION_BLOCK

(* POU FB_HARDWARE/FB_DEFAULT_AXISVALUE, ST *)
FUNCTION_BLOCK FB_DEFAULT_AXISVALUE
VAR_INPUT
	xDefaultValue:BOOL:=FALSE;
	sDeviceName:STRING(255);
END_VAR
VAR_OUTPUT
END_VAR
VAR_IN_OUT
	T_Axis:ST_AXIS;
END_VAR
VAR
END_VAR
(****************************************************************************************************************************************************)
(***********                                      This Functionblock set the default axis value for the Beckhoff drive                                         ************)
(****************************************************************************************************************************************************)
IF xDefaultValue THEN
	IF sDeviceName = 'Beckhoff' THEN
		CASE T_Axis.T_Config_Gen.iTyp OF
		(* linear axis Beckhoff *)
		1:	T_Axis.T_FileObj.sData[1]:='01:idxGrp:=16#4000;idxOff:=16#27;LEN:=16#8;Value:=200.0';(* Max velocity *)
			T_Axis.T_FileObj.sData[2]:='02:idxGrp:=16#4000;idxOff:=16#6;Len:=16#8;Value:=20.0';(* Vel Ref forward *)
			T_Axis.T_FileObj.sData[3]:='03:idxGrp:=16#4000;idxOff:=16#7;LEN:=16#8;Value:=20.0';(* Vel Ref backward *)
			T_Axis.T_FileObj.sData[4]:='04:idxGrp:=16#4000;idxOff:=16#101;Len:=16#8;Value:=3800.0';(* Acc *)
			T_Axis.T_FileObj.sData[5]:='05:idxGrp:=16#4000;idxOff:=16#102;Len:=16#8;Value:=3800.0';(* Dec *)
			T_Axis.T_FileObj.sData[6]:='06:idxGrp:=16#4000;idxOff:=16#103;Len:=16#8;Value:=80222.0';(* Jerk *)
			T_Axis.T_FileObj.sData[7]:='07:idxGrp:=16#4000;idxOff:=16#A;Len:=16#8;Value:=200.0';(* Rapid traverse vel *)
			T_Axis.T_FileObj.sData[8]:='08:idxGrp:=16#5000;idxOff:=16#B;Len:=16#2;Value:=0';(* Enable min soft pos *)
			T_Axis.T_FileObj.sData[9]:='09:idxGrp:=16#5000;idxOff:=16#D;Len:=16#8;Value:=0';(* Min soft pos *)
			T_Axis.T_FileObj.sData[10]:='10:idxGrp:=16#5000;idxOff:=16#C;Len:=16#2;Value:=0';(* Enable max soft pos *)
			T_Axis.T_FileObj.sData[11]:='11:idxGrp:=16#5000;idxOff:=16#E;Len:=16#8;Value:=0';(* Max soft pos *)
			T_Axis.T_FileObj.sData[12]:='12:idxGrp:=16#6000;idxOff:=16#10;Len:=16#2;Value:=1';(* Enable pos lag *)
			T_Axis.T_FileObj.sData[13]:='13:idxGrp:=16#6000;idxOff:=16#12;Len:=16#8;Value:=10.0';(* Max Pos lag *)
			T_Axis.T_FileObj.sData[14]:='14:idxGrp:=16#5000;idxOff:=16#8;Len:=16#2;Value:=0';(* Invert Enc counting *)
			T_Axis.T_FileObj.sData[15]:='15:idxGrp:=16#5000;idxOff:=16#6;Len:=16#8;Value:=3.81e-5';(* Enc scaling factor *)
			T_Axis.T_FileObj.sData[16]:='16:idxGrp:=16#5000;idxOff:=16#9;Len:=16#8;Value:=1';(* Enc modulo factor *)
			T_Axis.T_FileObj.sData[17]:='17:idxGrp:=16#5000;idxOff:=16#101;Len:=16#2;Value:=1';(* Enc dir for ref search *)
			T_Axis.T_FileObj.sData[18]:='18:idxGrp:=16#5000;idxOff:=16#102;Len:=16#2;Value:=0';(* Enc dir for sync impuls*)
			T_Axis.T_FileObj.sData[19]:='19:idxGrp:=16#5000;idxOff:=16#103;Len:=16#8;Value:=0';(* Enc ref value *)
			T_Axis.T_FileObj.sData[20]:='20:idxGrp:=16#5000;idxOff:=16#106;Len:=16#2;Value:=0';(* Enc Ext sync impuls *)
			T_Axis.T_FileObj.sData[21]:='21:idxGrp:=16#5000;idxOff:=16#107;Len:=16#4;Value:=5';(* Enc ref sequence *)
			T_Axis.T_FileObj.sData[22]:='22:idxGrp:=16#7000;idxOff:=16#6;Len:=16#2;Value:=0';(* Driver invert polarity *)
			T_Axis.T_FileObj.sData[23]:='23:idxGrp:=16#7000;idxOff:=16#101;Len:=16#8;Value:=220';(* Driver Max Ref vel *)
			T_Axis.T_FileObj.sData[24]:='24:idxGrp:=16#7000;idxOff:=16#102;Len:=16#8;Value:=0.75';(* Driver output ration *)
			T_Axis.T_FileObj.sData[25]:='25:idxGrp:=16#6000;idxOff:=16#B;Len:=16#8;Value:=1';(* Ctrler pre-ctrl weighting *)
			T_Axis.T_FileObj.sData[26]:='26:idxGrp:=16#6000;idxOff:=16#102;LEN:=16#8;Value:=50';(* Ctrler Kv factor *)
			T_Axis.T_FileObj.sData[27]:='';
		(* spindle axis Beckhoff *)
		2:	T_Axis.T_FileObj.sData[1]:='01:idxGrp:=16#4000;idxOff:=16#27;LEN:=16#8;Value:=24000.0';(* Max velocity *)
			T_Axis.T_FileObj.sData[2]:='02:idxGrp:=16#4000;idxOff:=16#6;Len:=16#8;Value:=60.0';(* Vel Ref forward *)
			T_Axis.T_FileObj.sData[3]:='03:idxGrp:=16#4000;idxOff:=16#7;LEN:=16#8;Value:=60.0';(* Vel Ref backward *)
			T_Axis.T_FileObj.sData[4]:='04:idxGrp:=16#4000;idxOff:=16#101;Len:=16#8;Value:=42000.0';(* Acc *)
			T_Axis.T_FileObj.sData[5]:='05:idxGrp:=16#4000;idxOff:=16#102;Len:=16#8;Value:=42000.0';(* Dec *)
			T_Axis.T_FileObj.sData[6]:='06:idxGrp:=16#4000;idxOff:=16#103;Len:=16#8;Value:=98000.0';(* Jerk *)
			T_Axis.T_FileObj.sData[7]:='07:idxGrp:=16#4000;idxOff:=16#A;Len:=16#8;Value:=24000.0';(* Rapid traverse vel *)
			T_Axis.T_FileObj.sData[8]:='08:idxGrp:=16#5000;idxOff:=16#B;Len:=16#2;Value:=0';(* Enable min soft pos *)
			T_Axis.T_FileObj.sData[9]:='09:idxGrp:=16#5000;idxOff:=16#D;Len:=16#8;Value:=0';(* Min soft pos *)
			T_Axis.T_FileObj.sData[10]:='10:idxGrp:=16#5000;idxOff:=16#C;Len:=16#2;Value:=0';(* Enable max soft pos *)
			T_Axis.T_FileObj.sData[11]:='11:idxGrp:=16#5000;idxOff:=16#E;Len:=16#8;Value:=0';(* Max soft pos *)
			T_Axis.T_FileObj.sData[12]:='12:idxGrp:=16#6000;idxOff:=16#10;Len:=16#2;Value:=1';(* Enable pos lag *)
			T_Axis.T_FileObj.sData[13]:='13:idxGrp:=16#6000;idxOff:=16#12;Len:=16#8;Value:=90.0';(* Max Pos lag *)
			T_Axis.T_FileObj.sData[14]:='14:idxGrp:=16#5000;idxOff:=16#8;Len:=16#2;Value:=0';(* Invert Enc counting *)
			T_Axis.T_FileObj.sData[15]:='15:idxGrp:=16#5000;idxOff:=16#6;Len:=16#8;Value:=0.00549';(* Enc scaling factor *)
			T_Axis.T_FileObj.sData[16]:='16:idxGrp:=16#5000;idxOff:=16#9;Len:=16#8;Value:=360';(* Enc modulo factor *)
			T_Axis.T_FileObj.sData[17]:='17:idxGrp:=16#5000;idxOff:=16#101;Len:=16#2;Value:=1';(* Enc dir for ref search *)
			T_Axis.T_FileObj.sData[18]:='18:idxGrp:=16#5000;idxOff:=16#102;Len:=16#2;Value:=0';(* Enc dir for sync impuls*)
			T_Axis.T_FileObj.sData[19]:='19:idxGrp:=16#5000;idxOff:=16#103;Len:=16#8;Value:=0';(* Enc ref value *)
			T_Axis.T_FileObj.sData[20]:='20:idxGrp:=16#5000;idxOff:=16#106;Len:=16#2;Value:=0';(* Enc Ext sync impuls *)
			T_Axis.T_FileObj.sData[21]:='21:idxGrp:=16#5000;idxOff:=16#107;Len:=16#4;Value:=5';(* Enc ref sequence *)
			T_Axis.T_FileObj.sData[22]:='22:idxGrp:=16#7000;idxOff:=16#6;Len:=16#2;Value:=0';(* Driver invert polarity *)
			T_Axis.T_FileObj.sData[23]:='23:idxGrp:=16#7000;idxOff:=16#101;Len:=16#8;Value:=26000';(* Driver Max Ref vel *)
			T_Axis.T_FileObj.sData[24]:='24:idxGrp:=16#7000;idxOff:=16#102;Len:=16#8;Value:=1';(* Driver output ration *)
			T_Axis.T_FileObj.sData[25]:='25:idxGrp:=16#6000;idxOff:=16#B;Len:=16#8;Value:=1';(* Ctrler pre-ctrl weighting *)
			T_Axis.T_FileObj.sData[26]:='26:idxGrp:=16#6000;idxOff:=16#102;LEN:=16#8;Value:=0.5';(* Ctrler Kv factor *)
			T_Axis.T_FileObj.sData[27]:='';
		(* spindle axis Beckhoff *)
		3:	T_Axis.T_FileObj.sData[1]:='01:idxGrp:=16#4000;idxOff:=16#27;LEN:=16#8;Value:=24000.0';(* Max velocity *)
			T_Axis.T_FileObj.sData[2]:='02:idxGrp:=16#4000;idxOff:=16#6;Len:=16#8;Value:=60.0';(* Vel Ref forward *)
			T_Axis.T_FileObj.sData[3]:='03:idxGrp:=16#4000;idxOff:=16#7;LEN:=16#8;Value:=60.0';(* Vel Ref backward *)
			T_Axis.T_FileObj.sData[4]:='04:idxGrp:=16#4000;idxOff:=16#101;Len:=16#8;Value:=42000.0';(* Acc *)
			T_Axis.T_FileObj.sData[5]:='05:idxGrp:=16#4000;idxOff:=16#102;Len:=16#8;Value:=42000.0';(* Dec *)
			T_Axis.T_FileObj.sData[6]:='06:idxGrp:=16#4000;idxOff:=16#103;Len:=16#8;Value:=98000.0';(* Jerk *)
			T_Axis.T_FileObj.sData[7]:='07:idxGrp:=16#4000;idxOff:=16#A;Len:=16#8;Value:=24000.0';(* Rapid traverse vel *)
			T_Axis.T_FileObj.sData[8]:='08:idxGrp:=16#5000;idxOff:=16#B;Len:=16#2;Value:=0';(* Enable min soft pos *)
			T_Axis.T_FileObj.sData[9]:='09:idxGrp:=16#5000;idxOff:=16#D;Len:=16#8;Value:=0';(* Min soft pos *)
			T_Axis.T_FileObj.sData[10]:='10:idxGrp:=16#5000;idxOff:=16#C;Len:=16#2;Value:=0';(* Enable max soft pos *)
			T_Axis.T_FileObj.sData[11]:='11:idxGrp:=16#5000;idxOff:=16#E;Len:=16#8;Value:=0';(* Max soft pos *)
			T_Axis.T_FileObj.sData[12]:='12:idxGrp:=16#6000;idxOff:=16#10;Len:=16#2;Value:=1';(* Enable pos lag *)
			T_Axis.T_FileObj.sData[13]:='13:idxGrp:=16#6000;idxOff:=16#12;Len:=16#8;Value:=90.0';(* Max Pos lag *)
			T_Axis.T_FileObj.sData[14]:='14:idxGrp:=16#5000;idxOff:=16#8;Len:=16#2;Value:=0';(* Invert Enc counting *)
			T_Axis.T_FileObj.sData[15]:='15:idxGrp:=16#5000;idxOff:=16#6;Len:=16#8;Value:=0.00549';(* Enc scaling factor *)
			T_Axis.T_FileObj.sData[16]:='16:idxGrp:=16#5000;idxOff:=16#9;Len:=16#8;Value:=360';(* Enc modulo factor *)
			T_Axis.T_FileObj.sData[17]:='17:idxGrp:=16#5000;idxOff:=16#101;Len:=16#2;Value:=1';(* Enc dir for ref search *)
			T_Axis.T_FileObj.sData[18]:='18:idxGrp:=16#5000;idxOff:=16#102;Len:=16#2;Value:=0';(* Enc dir for sync impuls*)
			T_Axis.T_FileObj.sData[19]:='19:idxGrp:=16#5000;idxOff:=16#103;Len:=16#8;Value:=0';(* Enc ref value *)
			T_Axis.T_FileObj.sData[20]:='20:idxGrp:=16#5000;idxOff:=16#106;Len:=16#2;Value:=0';(* Enc Ext sync impuls *)
			T_Axis.T_FileObj.sData[21]:='21:idxGrp:=16#5000;idxOff:=16#107;Len:=16#4;Value:=5';(* Enc ref sequence *)
			T_Axis.T_FileObj.sData[22]:='22:idxGrp:=16#7000;idxOff:=16#6;Len:=16#2;Value:=1';(* Driver invert polarity *)
			T_Axis.T_FileObj.sData[23]:='23:idxGrp:=16#7000;idxOff:=16#101;Len:=16#8;Value:=26000';(* Driver Max Ref vel *)
			T_Axis.T_FileObj.sData[24]:='24:idxGrp:=16#7000;idxOff:=16#102;Len:=16#8;Value:=1';(* Driver output ration *)
			T_Axis.T_FileObj.sData[25]:='25:idxGrp:=16#6000;idxOff:=16#B;Len:=16#8;Value:=1';(* Ctrler pre-ctrl weighting *)
			T_Axis.T_FileObj.sData[26]:='26:idxGrp:=16#6000;idxOff:=16#102;LEN:=16#8;Value:=0.5';(* Ctrler Kv factor *)
			T_Axis.T_FileObj.sData[27]:='';
		END_CASE
	END_IF
END_IF
END_FUNCTION_BLOCK

(* POU FB_HARDWARE/FB_CONVERT_PARA_AXIS, ST *)
FUNCTION_BLOCK FB_CONVERT_PARA_AXIS
VAR_INPUT
	xStart:BOOL;
	iConversion:INT;
	sDeviceName:STRING(255);
END_VAR
VAR_IN_OUT
	T_Axis:ST_AXIS;
END_VAR
VAR_OUTPUT
	xDone:BOOL;
	xBusy:BOOL;
	xError:BOOL;
	diErrorNr:DINT;
END_VAR
VAR
(* trigger *)
	RisingEdgeStart:R_TRIG;
(* variable *)
	i: INT;
	iPosCarStart,iPosCarStop:INT;
	iStepConvertValueString:INT;
(* tmp variable *)
	sTmp:STRING(255);
	jj: INT;
END_VAR
(****************************************************************************************************************************************************)
(***********                                    This Functionblock convert the axis parameter for the Beckhoff drive                                       ************)
(****************************************************************************************************************************************************)
(* wait start *)
	RisingEdgeStart(CLK:=xStart);
	IF RisingEdgeStart.Q THEN
	(* init. varaible *)
		iStepConvertValueString:=1;
		xDone:=FALSE;
	(*activ busy flag*)
		xBusy:=TRUE;
		xError:=FALSE;
		diErrorNr:=0;
	END_IF

(* test if activ *)
	IF NOT(xBusy) THEN
	(* exit FB *)
		RETURN;
	END_IF
	IF iConversion = 0 THEN
	(* conversion string to value *)
		i:=1;
		(* read string line-->Group or NodeId *)
		sTmp:=T_Axis.T_FileObj.sData[i];
		iPosCarStart:=FIND(sTmp,':=')+2;
		iPosCarStop:=FIND(sTmp,';');
		IF ((iPosCarStart - 2) = 0) OR (iPosCarStop = 0) OR (iPosCarStart >= iPosCarStop) THEN xBusy:=FALSE;	xDone:=FALSE; xError:=TRUE; diErrorNr:=16#F100;	(* Wrong Syntax from Axis File *) RETURN; END_IF;
		IF sDeviceName = 'Beckhoff' THEN
			T_Axis.T_Config_Gen.udiNC_TaskIdxGrp:=STRING_TO_UDINT(MID(sTmp,iPosCarStop-iPosCarStart,iPosCarStart));
			T_Axis.T_Config_Gen.udiNodeId:=0;
		END_IF;
		IF sDeviceName = 'Maxon' THEN
			T_Axis.T_Config_Gen.udiNC_TaskIdxGrp:=0;
			T_Axis.T_Config_Gen.udiNodeId:=STRING_TO_UDINT(MID(sTmp,iPosCarStop-iPosCarStart,iPosCarStart));
		END_IF;
		i:=i+1;
		(* read string line-->ADS NetID *)
		sTmp:=T_Axis.T_FileObj.sData[i];
		iPosCarStart:=FIND(sTmp,':=')+2;
		iPosCarStop:=FIND(sTmp,';');
		IF ((iPosCarStart - 2) = 0) OR (iPosCarStop = 0) OR (iPosCarStart >= iPosCarStop) THEN xBusy:=FALSE;	xDone:=FALSE; xError:=TRUE; diErrorNr:=16#F100;	(* Wrong Syntax from Axis File *) RETURN; END_IF;
		IF sDeviceName = 'Beckhoff' THEN
			T_Axis.T_Config_Gen.sServoNetId:=MID(sTmp,iPosCarStop-iPosCarStart,iPosCarStart);
			T_Axis.T_Config_Gen.sAmsNetId:='';
		END_IF;
		IF sDeviceName = 'Maxon' THEN
			T_Axis.T_Config_Gen.sServoNetId:='';
			T_Axis.T_Config_Gen.sAmsNetId:=MID(sTmp,iPosCarStop-iPosCarStart,iPosCarStart);
		END_IF;
		i:=i+1;
		(* read string line-->DeviceName *)
		sTmp:=T_Axis.T_FileObj.sData[i];
		iPosCarStart:=FIND(sTmp,':=')+2;
   		iPosCarStop:=FIND(sTmp,';');
		IF ((iPosCarStart - 2) = 0) OR (iPosCarStop = 0) OR (iPosCarStart >= iPosCarStop) THEN xBusy:=FALSE;	xDone:=FALSE; xError:=TRUE; diErrorNr:=16#F100;	(* Wrong Syntax from Axis File *) RETURN; END_IF;
		T_Axis.T_Config_Gen.sDeviceFileName:=MID(sTmp,iPosCarStop-iPosCarStart,iPosCarStart);
		i:=i+1;
		IF sDeviceName = 'Beckhoff' THEN
			(* read string line-->Quickstop ramp deceleration *)
			sTmp:=T_Axis.T_FileObj.sData[i];
			iPosCarStart:=FIND(sTmp,':=')+2;
	   		iPosCarStop:=FIND(sTmp,';');
			IF ((iPosCarStart - 2) = 0) OR (iPosCarStop = 0) OR (iPosCarStart >= iPosCarStop) THEN xBusy:=FALSE;	xDone:=FALSE; xError:=TRUE; diErrorNr:=16#F100;	(* Wrong Syntax from Axis File *) RETURN; END_IF;
			T_Axis.T_Config_Setting.rHCRampDeceleration:=STRING_TO_REAL(MID(sTmp,iPosCarStop-iPosCarStart,iPosCarStart));
			i:=i+1;
			(* read string line-->Quickstop ramp jerk *)
			sTmp:=T_Axis.T_FileObj.sData[i];
			iPosCarStart:=FIND(sTmp,':=')+2;
	   		iPosCarStop:=FIND(sTmp,';');
			IF ((iPosCarStart - 2) = 0) OR (iPosCarStop = 0) OR (iPosCarStart >= iPosCarStop) THEN xBusy:=FALSE;	xDone:=FALSE; xError:=TRUE; diErrorNr:=16#F100;	(* Wrong Syntax from Axis File *) RETURN; END_IF;
			T_Axis.T_Config_Setting.rHCRampJerk:=STRING_TO_REAL(MID(sTmp,iPosCarStop-iPosCarStart,iPosCarStart));
			i:=i+1;
		END_IF;
		jj:=1;
		(* read string lines *)
		WHILE T_Axis.T_FileObj.sData[i] <> '' DO
			sTmp:=T_Axis.T_FileObj.sData[i];
			(* index group *)
			iPosCarStart:=FIND(sTmp,':=')+2;
			iPosCarStop:=FIND(sTmp,';');
			IF ((iPosCarStart - 2) = 0) OR (iPosCarStop = 0) OR (iPosCarStart >= iPosCarStop) THEN xBusy:=FALSE;	xDone:=FALSE; xError:=TRUE; diErrorNr:=16#F100;	(* Wrong Syntax from Axis File *) RETURN; END_IF;
			T_Axis.T_ParamFileObj[jj].udiIdxGroup:=	STRING_TO_UDINT(MID(sTmp,iPosCarStop-iPosCarStart,iPosCarStart))
											+ T_Axis.T_Config_Gen.udiNC_TaskIdxGrp;
			sTmp:=MID(sTmp,LEN(sTmp)-iPosCarStop, iPosCarStop+1);
			(* index offset *)
			iPosCarStart:=FIND(sTmp,':=')+2;
			iPosCarStop:=FIND(sTmp,';');
			IF ((iPosCarStart - 2) = 0) OR (iPosCarStop = 0) OR (iPosCarStart >= iPosCarStop) THEN xBusy:=FALSE;	xDone:=FALSE; xError:=TRUE; diErrorNr:=16#F100;	(* Wrong Syntax from Axis File *) RETURN; END_IF;
			T_Axis.T_ParamFileObj[jj].udiIndexOffset:=STRING_TO_UDINT(MID(sTmp,iPosCarStop-iPosCarStart,iPosCarStart));
			sTmp:=MID(sTmp,LEN(sTmp)-iPosCarStop, iPosCarStop+1);
			(* length value *)
			iPosCarStart:=FIND(sTmp,':=')+2;
			iPosCarStop:=FIND(sTmp,';');
			IF ((iPosCarStart - 2) = 0) OR (iPosCarStop = 0) OR (iPosCarStart >= iPosCarStop) THEN xBusy:=FALSE;	xDone:=FALSE; xError:=TRUE; diErrorNr:=16#F100;	(* Wrong Syntax from Axis File *) RETURN; END_IF;
			T_Axis.T_ParamFileObj[jj].udiLength:=STRING_TO_UDINT(MID(sTmp,iPosCarStop-iPosCarStart,iPosCarStart));
			sTmp:=MID(sTmp,LEN(sTmp)-iPosCarStop, iPosCarStop+1);
			(* value*)
			iPosCarStart:=FIND(sTmp,':=')+2;
			iPosCarStop:=FIND(sTmp,';');
			IF ((iPosCarStart - 2) = 0) OR (iPosCarStop = 0) OR (iPosCarStart >= iPosCarStop) THEN xBusy:=FALSE;	xDone:=FALSE; xError:=TRUE; diErrorNr:=16#F100;	(* Wrong Syntax from Axis File *) RETURN; END_IF;
			T_Axis.T_ParamFileObj[jj].lrReal:=STRING_TO_REAL(MID(sTmp,iPosCarStop-iPosCarStart,iPosCarStart));
			(* init existing line, erase text *)
			iPosCarStop:=FIND(T_Axis.T_FileObj.sData[i],'(');
			T_Axis.T_FileObj.sData[i]:=MID(T_Axis.T_FileObj.sData[i],iPosCarStop-1,1);
			(* next line *)
			i:=i+1;
			jj:=jj+1;
		END_WHILE
		(* init. next *)
		T_Axis.T_ParamFileObj[jj].udiIdxGroup:=0;
		T_Axis.T_ParamFileObj[jj].udiIndexOffset:=0;
		T_Axis.T_ParamFileObj[jj].udiLength:=0;
		T_Axis.T_ParamFileObj[jj].lrReal:=0;

	(* Init. NC parameter *)
		i:=1;
		(* Beckhoff *)
		IF sDeviceName = 'Beckhoff' THEN
			(*copy parameter value *)
			WHILE T_Axis.T_ParamFileObj[i].udiIdxGroup <> 0 DO
				CASE (T_Axis.T_ParamFileObj[i].udiIdxGroup - T_Axis.T_Config_Gen.udiNC_TaskIdxGrp) OF
				16#4000:	CASE T_Axis.T_ParamFileObj[i].udiIndexOffset OF
						(* Calibration velocity forward *)
						16#6:	T_Axis.T_Config_ObjFileValue.lrCalVelocityForward:=T_Axis.T_ParamFileObj[i].lrReal;
						(* Calibration velocity backward *)
						16#7:	T_Axis.T_Config_ObjFileValue.lrCalVelocityBackward:=T_Axis.T_ParamFileObj[i].lrReal;
						(* Maximum velocity *)
						16#27:	T_Axis.T_Config_ObjFileValue.lrMaxVelocity:=T_Axis.T_ParamFileObj[i].lrReal;
						(* Acceleration *)
						16#101:	T_Axis.T_Config_ObjFileValue.lrAcceleration:=T_Axis.T_ParamFileObj[i].lrReal;
						(* Decceleration *)
						16#102:	T_Axis.T_Config_ObjFileValue.lrDecceleration:=T_Axis.T_ParamFileObj[i].lrReal;
						(* Jerk *)
						16#103:	T_Axis.T_Config_ObjFileValue.lrJerk:=T_Axis.T_ParamFileObj[i].lrReal;
						END_CASE
				16#5000:	CASE T_Axis.T_ParamFileObj[i].udiIndexOffset OF
						(* Encoder scaling factor *)
						16#6:	T_Axis.T_Config_ObjFileValue.lrScaleFactor:=T_Axis.T_ParamFileObj[i].lrReal;
						(* SW limit negativ On/Off *)
						16#B:	T_Axis.T_Config_ObjFileValue.xSWLimitNeg:=REAL_TO_BOOL(T_Axis.T_ParamFileObj[i].lrReal);
						(* SW limit positiv On/Off *)
						16#C:	T_Axis.T_Config_ObjFileValue.xSWLimitPos:=REAL_TO_BOOL(T_Axis.T_ParamFileObj[i].lrReal);
						(* SW limit negativ value *)
						16#D:	T_Axis.T_Config_ObjFileValue.lrSWLimitNeg:=T_Axis.T_ParamFileObj[i].lrReal;
						(* SW limit position value *)
						16#E:	T_Axis.T_Config_ObjFileValue.lrSWLimitPos:=T_Axis.T_ParamFileObj[i].lrReal;
						END_CASE
				16#6000:;
				16#7000:;
				END_CASE
				(* next parameter *)
				i:=i+1;
			END_WHILE
		END_IF

		(* Maxon *)
		IF sDeviceName = 'Maxon' THEN
			(*copy parameter value *)
			WHILE T_Axis.T_ParamFileObj[i].udiIdxGroup <> 0 DO
				CASE T_Axis.T_ParamFileObj[i].udiIdxGroup  OF
				16#6083:	CASE T_Axis.T_ParamFileObj[i].udiIndexOffset OF
						(* Acceleration *)
						16#0:	T_Axis.T_Config_ObjFileValue.lrAcceleration:=T_Axis.T_ParamFileObj[i].lrReal;
						END_CASE
				16#6084:	CASE T_Axis.T_ParamFileObj[i].udiIndexOffset OF
						(* Decceleration *)
						16#0:	T_Axis.T_Config_ObjFileValue.lrDecceleration:=T_Axis.T_ParamFileObj[i].lrReal;
						END_CASE
				END_CASE
				(* next parameter *)
				i:=i+1;
			END_WHILE
		END_IF
		(* set flag done *)
		xBusy:=FALSE;
		xDone:=TRUE;
	END_IF;
END_FUNCTION_BLOCK

(* POU FB_HARDWARE/FBHW_AXIS_LIVEVALUES_BECKHOFF, ST *)
FUNCTION_BLOCK FBHW_AXIS_LIVEVALUES_BECKHOFF
VAR_INPUT
	uiActualTorque: UINT;
	arxDigitalInput: ARRAY[1..8] OF BOOL;
END_VAR
VAR_OUTPUT
END_VAR
VAR_IN_OUT
	T_Axis:ST_AXIS;
	T_AxisRefIn:NCTOPLC_AXLESTRUCT;
END_VAR
VAR
	i:INT;
END_VAR
(****************************************************************************************************************************************************)
(***********                                    This Functionblock read the actual value from the Beckhoff drive                                               ************)
(****************************************************************************************************************************************************)
(* return actual axis state *)
T_Axis.T_LiveValue.dwState:=T_AxisRefIn.nStateDWord;
(* return actual torque value *)
T_Axis.T_LiveValue.uiActualTorque:=uiActualTorque;
IF T_Axis.T_LiveValue.uiActualTorque > 16#7FFF THEN
	(* negativ value *)
	T_Axis.T_LiveValue.diActualTorqueCalc:=UINT_TO_DINT(T_Axis.T_LiveValue.uiActualTorque) - 65535;
ELSE
	(* positiv value *)
	T_Axis.T_LiveValue.diActualTorqueCalc:=UINT_TO_DINT(T_Axis.T_LiveValue.uiActualTorque);
END_IF
(* return actual velocity *)
T_Axis.T_LiveValue.lrActualVelocity:=T_AxisRefIn.fVeloIst;
(* ??? modif 06092005 *)
(* return actual position *)
IF T_Axis.T_Config_Gen.iTyp <>1 THEN
(* modulo position for rotativ axis*)
	T_Axis.T_LiveValue.lrActualPosition:=T_AxisRefIn.fModuloPosIst;
	T_Axis.T_LiveValue.lrActualPositionNotModulo:=T_AxisRefIn.fPosIst;
ELSE
(* counter value *)
	T_Axis.T_LiveValue.lrActualPosition:=T_AxisRefIn.fPosIst;
END_IF
T_Axis.T_LiveValue.lrSollPosition:=T_AxisRefIn.fPosSoll;
(* return actual position *)
(*T_Axis.T_LiveValue.lrActualPosition:=T_AxisRefIn.fPosIst;*)
(* ??? modif 06092005 *)
(* return the actual digital input state *)
T_Axis.T_LiveValue.bDigitalInput:=0;
FOR i := 0 TO 7 DO
	IF arxDigitalInput[i+1] THEN
		T_Axis.T_LiveValue.bDigitalInput:=T_Axis.T_LiveValue.bDigitalInput + MUX(i,1,2,4,8,16,32,64,128);
	END_IF
END_FOR;
END_FUNCTION_BLOCK

(* POU FB_HARDWARE/FBHW_AXIS_MULTI_BECKHOFF, ST *)
FUNCTION_BLOCK FBHW_AXIS_MULTI_BECKHOFF
VAR_INPUT
END_VAR
VAR_OUTPUT
END_VAR
VAR_IN_OUT
	T_AxisMaster:ST_AXIS;
	T_AxisSlave:ST_AXIS;
	T_AxisMasterRefIn:NCTOPLC_AXLESTRUCT;
	T_AxisSlaveRefIn:NCTOPLC_AXLESTRUCT;
END_VAR
VAR
(* block function *)
	fbAxisMasterSlaveOn:MC_GearIn;
	fbAxisMasterSlaveOff:MC_GearOut;
(* variable *)
	xGearIn:BOOL:=FALSE;
	xGearOut:BOOL:=FALSE;
	xConfirmResetFB:BOOL:=FALSE;
(* trigger *)
	RisingEdgeResetFB:R_TRIG;
	RisingEdgeExecute:R_TRIG;
END_VAR
(****************************************************************************************************************************************************)
(***********                                   This Functionblock is the driver for the Beckhoff Axis for Master/Slave                                      ************)
(****************************************************************************************************************************************************)
(* Reset block function *)
	RisingEdgeResetFB(CLK:=T_AxisMaster.T_CtrleMulti.xReset);
	IF RisingEdgeResetFB.Q THEN
	(* Init. block function *)
		fbAxisMasterSlaveOn(	Execute:=FALSE,
							Master:=T_AxisMasterRefIn,
							Slave:=T_AxisSlaveRefIn);
		fbAxisMasterSlaveOff(	Execute:=FALSE,
							Slave:=T_AxisSlaveRefIn);
	(* Init. variable *)
		xGearIn:=FALSE;
		xGearOut:=FALSE;
	(* init. structure *)
		T_AxisMaster.T_CtrleMulti.iFunction:=0;
		T_AxisMaster.T_CtrleMulti.iNumerator:=1;
		T_AxisMaster.T_CtrleMulti.uiDenominator:=1;
		T_AxisMaster.T_CtrleMulti.xDone:=FALSE;
		T_AxisMaster.T_CtrleMulti.xErr:=FALSE;
		T_AxisMaster.T_CtrleMulti.udiErrorID:=0;
		(* set done flag *)
		xConfirmResetFB:=TRUE;
		(* exit function bloc *)
		RETURN;
	ELSE
		IF xConfirmResetFB THEN
		(* confirm reset FB *)
			T_AxisMaster.T_CtrleMulti.xDone:=TRUE;
			T_AxisMaster.T_CtrleMulti.xErr:=FALSE;
			T_AxisMaster.T_CtrleMulti.udiErrorID:=0;
			(* reset variable *)
			xConfirmResetFB:=FALSE;
		END_IF
	END_IF

(* Execute *)
	RisingEdgeExecute(CLK:=T_AxisMaster.T_CtrleMulti.xExecute);
	IF RisingEdgeExecute.Q THEN
		CASE T_AxisMaster.T_CtrleMulti.iFunction OF
		(* activ master-slave *)
		1:	xGearIn:=TRUE;
		(* desactiv master-slave *)
		2: 	xGearOut:=TRUE;
		ELSE
		(* function not implemented *)
			T_AxisMaster.T_CtrleMulti.xDone:=FALSE;
			T_AxisMaster.T_CtrleMulti.xErr:=TRUE;
			T_AxisMaster.T_CtrleMulti.udiErrorID:=16#F000;
			(* exit FB *)
			RETURN;
		END_CASE
		(* Init. variable *)
		T_AxisMaster.T_CtrleMulti.xDone:=FALSE;
		T_AxisMaster.T_CtrleMulti.xErr:=FALSE;
		T_AxisMaster.T_CtrleMulti.udiErrorID:=0;
	END_IF

(* GearIn *)
	IF xGearIn THEN
		fbAxisMasterSlaveOn(	Execute:=TRUE,
							RatioNumerator:=T_AxisMaster.T_CtrleMulti.iNumerator,
							RatioDenominator:=T_AxisMaster.T_CtrleMulti.uiDenominator,
							Acceleration:=T_AxisMaster.T_CtrleSingle.lrAcceleration,
							Deceleration:=T_AxisMaster.T_CtrleSingle.lrDecceleration,
							Jerk:=T_AxisMaster.T_CtrleSingle.lrJerk,
							Master:=T_AxisMasterRefIn,
							Slave:=T_AxisSlaveRefIn);
		IF fbAxisMasterSlaveOn.InGear OR fbAxisMasterSlaveOn.Error THEN
			T_AxisMaster.T_CtrleMulti.xDone:= fbAxisMasterSlaveOn.InGear;
			T_AxisMaster.T_CtrleMulti.xErr:=fbAxisMasterSlaveOn.Error;
			T_AxisMaster.T_CtrleMulti.udiErrorID:=fbAxisMasterSlaveOn.ErrorID;
			(* set flag gearin off *)
			xGearIn:=FALSE;
		END_IF
	ELSE
		fbAxisMasterSlaveOn(	Execute:=FALSE,
							Master:=T_AxisMasterRefIn,
							Slave:=T_AxisSlaveRefIn);
	END_IF

(* GearOut *)
	IF xGearOut THEN
		fbAxisMasterSlaveOff(	Execute:=TRUE,
							Slave:=T_AxisSlaveRefIn);
		IF fbAxisMasterSlaveOff.Done OR fbAxisMasterSlaveOff.Error THEN
			T_AxisMaster.T_CtrleMulti.xDone:= fbAxisMasterSlaveOff.Done;
			T_AxisMaster.T_CtrleMulti.xErr:=fbAxisMasterSlaveOff.Error;
			T_AxisMaster.T_CtrleMulti.udiErrorID:=fbAxisMasterSlaveOff.ErrorID;
			(* set flag gearout off *)
			xGearOut:=FALSE;
		END_IF
	ELSE
		fbAxisMasterSlaveOff(	Execute:=FALSE,
							Slave:=T_AxisSlaveRefIn);
	END_IF
END_FUNCTION_BLOCK

(* POU FB_HARDWARE/FBHW_CYL_ANALOGCYLINDER, ST *)
FUNCTION_BLOCK FBHW_CYL_ANALOGCYLINDER
VAR_INPUT
	xCtrlePosOn:BOOL;
	xCtrlePosOff:BOOL;
	iAnalogIn:INT;
END_VAR
VAR_OUTPUT
	xCylinder:BOOL;
	iAnalogOut:INT;
END_VAR
VAR_IN_OUT
	T_Cylinder:ST_CYLINDER;
END_VAR
VAR
(* variable *)
	xConfirmResetFB: BOOL;
	xActivCtrle:BOOL;
	iStep:INT;
(* timer *)
	TimerOn:TON;
	TimerOff:TON;
	TimerPreOn:TON;
	TimerPreOff:TON;
	TimerOut:TON;
	TimerActiv: TON;
(* trigger *)
	RisingEdgeExecute:R_TRIG;
	RisingEdgeReset:R_TRIG;
	RisingEdgeActiv:R_TRIG;
	FallingEdgeActiv:F_TRIG;
	xFct3Activ: BOOL;
	xTmpFct3Activ: BOOL;
END_VAR
(****************************************************************************************************************************************************)
(***********                                       This Functionblock is the driver for the ToolTension Cylinder                                                    ************)
(****************************************************************************************************************************************************)
(* if function bloc set activ then Analog state will be transfered *)
	RisingEdgeActiv(CLK:=T_Cylinder.T_CtrleCyl.xFBActiv);
	FallingEdgeActiv(CLK:=T_Cylinder.T_CtrleCyl.xFBActiv);
	IF RisingEdgeActiv.Q OR FallingEdgeActiv.Q THEN
		iAnalogOut:=0;
		xCylinder:=NOT(T_Cylinder.T_Config.xActivState);
		T_Cylinder.T_CtrleCyl.T_AnalogCylinder.xActiv:= FALSE;
	END_IF
	(* transfer sensor state only if fb is activ *)
	IF T_Cylinder.T_CtrleCyl.xFBActiv THEN
		T_Cylinder.T_CtrleCyl.xStatePosOn:=xCtrlePosOn;
		T_Cylinder.T_CtrleCyl.xStatePosOff:=xCtrlePosOff;
	(* copy state value *)
		T_Cylinder.T_CtrleCyl.T_AnalogCylinder.iAnalogOut:=iAnalogOut;
	ELSE
	(* exit fb *)
		RETURN;
	END_IF

(* wait for reseting *)
	RisingEdgeReset(CLK:=T_Cylinder.T_CtrleCyl.xReset);
	IF RisingEdgeReset.Q THEN
		(* Init. timer *)
		TimerOn(IN:=TRUE,PT:=T#1ms);
		TimerOff(IN:=TRUE,PT:=T#1ms);
		TimerOut(IN:=TRUE,PT:=T#1ms);
		TimerPreOn(IN:=TRUE,PT:=T#1ms);
		TimerPreOff(IN:=TRUE,PT:=T#1ms);
		TimerActiv(IN:=TRUE,PT:=T#1ms);
	(* Init. variable *)
		xActivCtrle:=FALSE;
		iStep:=0;
		xFct3Activ:=FALSE;
		xTmpFct3Activ:=FALSE;
		T_Cylinder.T_CtrleCyl.T_AnalogCylinder.tDelayActiv:=T#0s;
		T_Cylinder.T_Config.tDelayPreOn:=T#0s;
		T_Cylinder.T_Config.tDelayPreOff:=T#0s;
	(* Init. structure *)
		T_Cylinder.T_CtrleCyl.iFunction:=0;
		T_Cylinder.T_CtrleCyl.T_AnalogCylinder.xActiv:= FALSE;
		xCylinder:=NOT(T_Cylinder.T_Config.xActivState);
		iAnalogOut:=0;
		T_Cylinder.T_CtrleCyl.xDone:=FALSE;
		T_Cylinder.T_CtrleCyl.xErr:=FALSE;
		T_Cylinder.T_CtrleCyl.udiErrorID:=16#0;
	(* confirm reset *)
		xConfirmResetFB:=TRUE;
	(* exit function *)
		RETURN;
	ELSE
		IF xConfirmResetFB THEN
		(* confirm reset FB *)
			T_Cylinder.T_CtrleCyl.xDone:=TRUE;
			T_Cylinder.T_CtrleCyl.xErr:=FALSE;
			T_Cylinder.T_CtrleCyl.udiErrorID:=16#0;
			(* init. variable *)
			xConfirmResetFB:=FALSE;
		END_IF
	END_IF

(* wait for execute *)
	RisingEdgeExecute(CLK:=T_Cylinder.T_CtrleCyl.xExecute);
	IF RisingEdgeExecute.Q THEN
		IF NOT(T_Cylinder.T_CtrleCyl.xDone) AND NOT(T_Cylinder.T_CtrleCyl.xErr) THEN
		(* can execute function if both signal are disable *)
			RETURN;
		END_IF
		CASE T_Cylinder.T_CtrleCyl.iFunction OF
		(* disable *)
		1:	iStep:=11;
		(* Activ without sensor position ctrle *)
		2:	iStep:=1;
		(* set value Analog Out = Analog In *)
		4:	iStep:=21;
		(* inverse cylinder state *)
		51:	iStep:=51;
		ELSE
			(* function not implemented *)
			iStep:=0;
			T_Cylinder.T_CtrleCyl.xDone:=FALSE;
			T_Cylinder.T_CtrleCyl.xErr:=TRUE;
			T_Cylinder.T_CtrleCyl.udiErrorID:=16#F000;
			(* exit FB *)
			RETURN;
		END_CASE
		(* Init. variable *)
		T_Cylinder.T_CtrleCyl.xDone:=FALSE;
		T_Cylinder.T_CtrleCyl.xErr:=FALSE;
		T_Cylinder.T_CtrleCyl.udiErrorID:=16#0;
		(* exit FB *)
		RETURN;
	END_IF

(* Timer activ *)
	TimerOn(IN:=TRUE,PT:=T_Cylinder.T_Config.tDelayOn);
	TimerOff(IN:=TRUE,PT:=T_Cylinder.T_Config.tDelayOff);
	TimerPreOn(IN:=TRUE,PT:=T_Cylinder.T_Config.tDelayPreOn);
	TimerPreOff(IN:=TRUE,PT:=T_Cylinder.T_Config.tDelayPreOff);
	TimerOut(IN:=TRUE,PT:=T_Cylinder.T_Config.tTimeOut);
	TimerActiv(IN:=TRUE,PT:=T_Cylinder.T_CtrleCyl.T_AnalogCylinder.tDelayActiv);
(* waiting for activ *)
	CASE iStep OF
	(* Set Analog output *)
	1:	IF (T_Cylinder.T_Config.tDelayPreOn = T#0s) THEN
			TimerOn(IN:=FALSE);
			iAnalogOut:=iAnalogIn;
			xCylinder:=T_Cylinder.T_Config.xActivState;
			T_Cylinder.T_CtrleCyl.T_AnalogCylinder.xActiv:= TRUE;
			iStep:=2;
		ELSE
			TimerPreOn(IN:=FALSE);
			iStep:=4;
		END_IF;
	(* wait for timer On *)
	2:	IF TimerOn.Q THEN
			iStep:=3;
			TimerOut(IN:=FALSE);
		END_IF
	(* control position activ *)
	3:	IF T_Cylinder.T_Config.xCtrlePosOn THEN
		(* position ctrle activ *)
			IF TimerOut.Q THEN
			(* timerout done, activ error cylinder has not activ position reached *)
				iStep:=999;
			ELSE
				IF xCtrlePosOn THEN
				(* Activ position reached, activ confirmation *)
					iStep:=90;
				END_IF
			END_IF
		ELSE
		(* no position ctrle, activ confirm *)
			iStep:=90;
		END_IF
	(* wait for timer Pre On *)
	4:	IF TimerPreOn.Q THEN
			T_Cylinder.T_Config.tDelayPreOn:=T#0s;
			iStep:=1;
		END_IF
	(* process timer Off *)
	11:	IF (T_Cylinder.T_Config.tDelayPreOff = T#0s) THEN
			TimerOff(IN:=FALSE);
			iAnalogOut:=0;
			xCylinder:=NOT(T_Cylinder.T_Config.xActivState);
			T_Cylinder.T_CtrleCyl.T_AnalogCylinder.xActiv:= FALSE;
			iStep:=12;
		ELSE
			TimerPreOff(IN:=FALSE);
			iStep:=14;
		END_IF;
	(* wait for timer Off *)
	12:	IF TimerOff.Q THEN
			iStep:=13;
			TimerOut(IN:=FALSE);
		END_IF
	(* control position inactiv *)
	13:	IF T_Cylinder.T_Config.xCtrlePosOff THEN
		(* control position activ *)
			IF TimerOut.Q THEN
			(* timerout done, activ error 'cylinder has not inactiv position reached' *)
				iStep:=998;
			ELSE
				IF xCtrlePosOff THEN
				(* inactiv position reached, activ confirmation *)
					iStep:=99;
				END_IF
			END_IF
		ELSE
		(* no control position activ, activ confirmation *)
			iStep:=99;
		END_IF
	(* wait for timer Pre Off *)
	14:	IF TimerPreOff.Q THEN
			T_Cylinder.T_Config.tDelayPreOff:=T#0s;
			iStep:=11;
		END_IF
	(* set value Analog Out = Analog In *)
	21:	xCylinder:=T_Cylinder.T_Config.xActivState;
		T_Cylinder.T_CtrleCyl.T_AnalogCylinder.xActiv:= TRUE;
		iAnalogOut:=iAnalogIn;
		iStep:=99;
	(* inverse cylinder state *)
	51:	IF T_Cylinder.T_CtrleCyl.T_AnalogCylinder.xActiv THEN
			iAnalogOut:=0;
		ELSE
			iAnalogOut:=iAnalogIn;
		END_IF;
		xCylinder:=NOT(xCylinder);
		T_Cylinder.T_CtrleCyl.T_AnalogCylinder.xActiv:=NOT(T_Cylinder.T_CtrleCyl.T_AnalogCylinder.xActiv);
		iStep:=99;
	(* test if delay activ *)
	90:	IF T_Cylinder.T_CtrleCyl.T_AnalogCylinder.tDelayActiv <> T#0s THEN
			TimerActiv(IN:=FALSE);
			iStep:=91;
		ELSE
			iStep:=99;
		END_IF
	(* wait for time delay activ *)
	91:	IF TimerActiv.Q THEN
			T_Cylinder.T_CtrleCyl.T_AnalogCylinder.tDelayActiv:=T#0s;
			iStep:=11;	(* Zylinder wird wieder deaktiviert *)
		END_IF;
	(* no ctrle position *)
	99:	T_Cylinder.T_CtrleCyl.xDone:=TRUE;
		T_Cylinder.T_CtrleCyl.xErr:=FALSE;
		T_Cylinder.T_CtrleCyl.udiErrorID:=16#0;
	(* error, cylinder not in inactiv position *)
	998:	T_Cylinder.T_CtrleCyl.xDone:=FALSE;
		T_Cylinder.T_CtrleCyl.xErr:=TRUE;
		T_Cylinder.T_CtrleCyl.udiErrorID:=16#F202;
	(* error, cylinder not in activ position *)
	999:	T_Cylinder.T_CtrleCyl.xDone:=FALSE;
		T_Cylinder.T_CtrleCyl.xErr:=TRUE;
		T_Cylinder.T_CtrleCyl.udiErrorID:=16#F201;
	END_CASE
END_FUNCTION_BLOCK

(* POU GENERAL/FB_CALC_TOOLTENSION_FORCE_NEW, ST *)
FUNCTION_BLOCK FB_CALC_TOOLTENSION_FORCE_NEW
VAR_INPUT
	rForcePistonIn:REAL;	(* in Newton *)
	rPistonDiameterD1:REAL;	(* in mm *)
	rPistonDiameterD2:REAL;	(* in mm *)
	rMaxAirpressure:REAL;		(* in bar *)
	rFactorForce:REAL;
END_VAR
VAR_OUTPUT
	iAnalogOutput:INT;		(* range 0 - 32767 *)
	rSetMaxForce:REAL;		(* in Newton *)
	rForcePistonOut:REAL;	(* in Newton *)
END_VAR
VAR
	rMaxForce: REAL;
	rAreaOutside: REAL;
	rAreaInside: REAL;
	rArea: REAL;
	rTmpMaxAirpressure: REAL;
	rTmpAnalogOut:REAL;
END_VAR
(****************************************************************************************************************************************************)
(*****       This Functionblock calculate the effective value for the servo ventil for the ToolTension which the settled force         *****)
(****************************************************************************************************************************************************)
	rAreaOutside:=((rPistonDiameterD1/2)*(rPistonDiameterD1/2))*PI;
	rAreaInside:=((rPistonDiameterD2/2)*(rPistonDiameterD2/2))*PI;
	rArea:=ABS(rAreaOutside - rAreaInside);
	rArea:=rArea / 1000000.0;	(* Umwandeln von mm^2 in m^2 *)
	rTmpMaxAirpressure:=rMaxAirpressure * 100000.0;	(* convert from bar to pascal *)
	rMaxForce:=rArea * rTmpMaxAirpressure * rFactorForce;
	rSetMaxForce:=rMaxForce;

	IF(rMaxForce = 0) THEN rMaxForce:=0.01; END_IF;	(* check divide by zero *)
	IF(rMaxForce <> 0.0) THEN
		rTmpAnalogOut:=(rForcePistonIn/rMaxForce)*32767;	(* 32767 = 10V *)
		IF (rTmpAnalogOut > 32767) THEN
			iAnalogOutput:=32767;
		ELSE
			iAnalogOutput:=REAL_TO_INT(rTmpAnalogOut);
		END_IF;
		rForcePistonOut:=rForcePistonIn;
	ELSE
		iAnalogOutput:=0;
		rForcePistonOut:=0;
	END_IF;
END_FUNCTION_BLOCK

